DATA_BLOCK "DB00800_St_K_AnData"   // DB800
TITLE = Static DB [CONSTANTS] — Analog Card Ranges, Types and Coefficients
{ S7_Optimized_Access := 'TRUE' }
AUTHOR : M_Gledhill
FAMILY : Constants
NAME : St_K_AnData
VERSION : 0.1
// PRACTICAL SERIES AUTOMATION LIBRARY (PAL)   —   COPYRIGHT 2020 – M. GLEDHILL (MIT LICENCE)
//                   ———— ◆ ————
// FULL ONLINE DOCUMENTATION IS AVAILABLE AT: https://practicalseries.com/2001-pal/index.html
// stored: AutoNumber false, DBAccessibleFromOPCUA true, IsOnlyStoredInLoadMemory false, IsRetainMemResEnabled false, IsWriteProtectedInAS true, MemoryReserve 100
   VAR
      _DB_Header { ExternalAccessible := 'False'; ExternalVisible := 'False'; ExternalWritable := 'False'} : Array[0..79] of Bool;   // Static DB [CONSTANTS] — Analog Card Ranges, Types and Coefficients
      __________0000_0 { ExternalAccessible := 'False'; ExternalVisible := 'False'; ExternalWritable := 'False'} : Bool := false;
      __________0000_1 { ExternalAccessible := 'False'; ExternalVisible := 'False'; ExternalWritable := 'False'} : Bool := false;   // ▀▀▀▀ DB CURRENT REVISION
      revInfo { ExternalWritable := 'False'; S7_SetPoint := 'True'} : "UT01000_St_SysRevision";   // Revision information
      __________0010_0 { ExternalAccessible := 'False'; ExternalVisible := 'False'; ExternalWritable := 'False'} : Bool := false;
      __________0010_1 { ExternalAccessible := 'False'; ExternalVisible := 'False'; ExternalWritable := 'False'} : Bool := false;   // ▀▀▀▀ ANALOG SIGNAL — USER DEFINED
      AIO_0000 : "UT00800_St_K_AnData";   // User defined signal type
      __________0020_0 { ExternalAccessible := 'False'; ExternalVisible := 'False'; ExternalWritable := 'False'} : Bool := false;
      __________0020_1 { ExternalAccessible := 'False'; ExternalVisible := 'False'; ExternalWritable := 'False'} : Bool := false;   // ▀▀▀▀ ANALOG SIGNAL — VOLTAGE
      AIO_1000 : "UT00800_St_K_AnData";   // Voltage (-25 mV to +25 mV)
      AIO_1001 : "UT00800_St_K_AnData";   // Voltage (-50 mV to +50 mV)
      AIO_1002 : "UT00800_St_K_AnData";   // Voltage (-80 mV to +80 mV)
      AIO_1003 : "UT00800_St_K_AnData";   // Voltage (-250 mV to +250 mV)
      AIO_1004 : "UT00800_St_K_AnData";   // Voltage (-500 mV to +500 mV)
      AIO_1005 : "UT00800_St_K_AnData";   // Voltage (-1 V to +1 V)
      AIO_1007 : "UT00800_St_K_AnData";   // Voltage (-2.5 V to +2.5 V)
      AIO_1008 : "UT00800_St_K_AnData";   // Voltage (-5 V to +5 V)
      AIO_1009 : "UT00800_St_K_AnData";   // Voltage (-10 V to +10 V)
      AIO_100A : "UT00800_St_K_AnData";   // Voltage (1 V to 5 V)
      __________0030_0 { ExternalAccessible := 'False'; ExternalVisible := 'False'; ExternalWritable := 'False'} : Bool := false;
      __________0030_1 { ExternalAccessible := 'False'; ExternalVisible := 'False'; ExternalWritable := 'False'} : Bool := false;   // ▀▀▀▀ ANALOG SIGNAL — CURRENT (4 WIRE)
      AIO_2002 : "UT00800_St_K_AnData";   // Current - 4 wire (0 mA to 20 mA)
      AIO_2003 : "UT00800_St_K_AnData";   // Current - 4 wire (4 mA to 20 mA)
      AIO_2004 : "UT00800_St_K_AnData";   // Current - 4 wire (-20 mA to +20 mA)
      __________0040_0 { ExternalAccessible := 'False'; ExternalVisible := 'False'; ExternalWritable := 'False'} : Bool := false;
      __________0040_1 { ExternalAccessible := 'False'; ExternalVisible := 'False'; ExternalWritable := 'False'} : Bool := false;   // ▀▀▀▀ ANALOG SIGNAL — CURRENT (2 WIRE)
      AIO_3003 : "UT00800_St_K_AnData";   // Current - 2 wire (4 mA to 20 mA)
      __________0050_0 { ExternalAccessible := 'False'; ExternalVisible := 'False'; ExternalWritable := 'False'} : Bool := false;
      __________0050_1 { ExternalAccessible := 'False'; ExternalVisible := 'False'; ExternalWritable := 'False'} : Bool := false;   // ▀▀▀▀ ANALOG SIGNAL — RESISTANCE (4 WIRE)
      AIO_4001 : "UT00800_St_K_AnData";   // Resistance - 4 wire (150 Ω)
      AIO_4002 : "UT00800_St_K_AnData";   // Resistance - 4 wire (300 Ohm)
      AIO_4003 : "UT00800_St_K_AnData";   // Resistance - 4 wire (600 Ohm)
      AIO_4005 : "UT00800_St_K_AnData";   // Resistance - 4 wire (6000 Ohm)
      __________0060_0 { ExternalAccessible := 'False'; ExternalVisible := 'False'; ExternalWritable := 'False'} : Bool := false;
      __________0060_1 { ExternalAccessible := 'False'; ExternalVisible := 'False'; ExternalWritable := 'False'} : Bool := false;   // ▀▀▀▀ ANALOG SIGNAL — RESISTANCE (3 WIRE)
      AIO_5001 : "UT00800_St_K_AnData";   // Resistance - 3 wire (150 Ohm)
      AIO_5002 : "UT00800_St_K_AnData";   // Resistance - 3 wire (300 Ohm)
      AIO_5003 : "UT00800_St_K_AnData";   // Resistance - 3 wire (600 Ohm)
      AIO_5005 : "UT00800_St_K_AnData";   // Resistance - 3 wire (6000 Ohm)
      __________0070_0 { ExternalAccessible := 'False'; ExternalVisible := 'False'; ExternalWritable := 'False'} : Bool := false;
      __________0070_1 { ExternalAccessible := 'False'; ExternalVisible := 'False'; ExternalWritable := 'False'} : Bool := false;   // ▀▀▀▀ ANALOG SIGNAL — RESISTANCE (2 WIRE)
      AIO_6001 : "UT00800_St_K_AnData";   // Resistance - 2 wire (150 Ohm)
      AIO_6002 : "UT00800_St_K_AnData";   // Resistance - 2 wire (300 Ohm)
      AIO_6003 : "UT00800_St_K_AnData";   // Resistance - 2 wire (600 Ohm)
      AIO_6005 : "UT00800_St_K_AnData";   // Resistance - 2 wire (6000 Ohm)
      AIO_600F : "UT00800_St_K_AnData";   // Resistance - 2 wire (PTC)
      __________0080_0 { ExternalAccessible := 'False'; ExternalVisible := 'False'; ExternalWritable := 'False'} : Bool := false;
      __________0080_1 { ExternalAccessible := 'False'; ExternalVisible := 'False'; ExternalWritable := 'False'} : Bool := false;   // ▀▀▀▀ ANALOG SIGNAL — THERMAL RESISTANCE (4 WIRE) Cu x0
      AIO_7B0E : "UT00800_St_K_AnData";   // Thermal Resistance - 4 wire (Cu10 climate - 426)
      AIO_7C0E : "UT00800_St_K_AnData";   // Thermal Resistance - 4 wire (Cu10 climate - 427)
      AIO_7D0E : "UT00800_St_K_AnData";   // Thermal Resistance - 4 wire (Cu10 climate - 428)
      AIO_7B0F : "UT00800_St_K_AnData";   // Thermal Resistance - 4 wire (Cu10 standard - 426)
      AIO_7C0F : "UT00800_St_K_AnData";   // Thermal Resistance - 4 wire (Cu10 standard - 427)
      AIO_7D0F : "UT00800_St_K_AnData";   // Thermal Resistance - 4 wire (Cu10 standard - 428)
      AIO_7B19 : "UT00800_St_K_AnData";   // Thermal Resistance - 4 wire (Cu50 climate - 426)
      AIO_7C19 : "UT00800_St_K_AnData";   // Thermal Resistance - 4 wire (Cu50 climate - 427)
      AIO_7D19 : "UT00800_St_K_AnData";   // Thermal Resistance - 4 wire (Cu50 climate - 428)
      AIO_7B18 : "UT00800_St_K_AnData";   // Thermal Resistance - 4 wire (Cu50 standard - 426)
      AIO_7C18 : "UT00800_St_K_AnData";   // Thermal Resistance - 4 wire (Cu50 standard - 427)
      AIO_7D18 : "UT00800_St_K_AnData";   // Thermal Resistance - 4 wire (Cu50 standard - 428)
      AIO_7B1B : "UT00800_St_K_AnData";   // Thermal Resistance - 4 wire (Cu100 climate - 426)
      AIO_7C1B : "UT00800_St_K_AnData";   // Thermal Resistance - 4 wire (Cu100 climate - 427)
      AIO_7D1B : "UT00800_St_K_AnData";   // Thermal Resistance - 4 wire (Cu100 climate - 428)
      AIO_7B1A : "UT00800_St_K_AnData";   // Thermal Resistance - 4 wire (Cu100 standard - 426)
      AIO_7C1A : "UT00800_St_K_AnData";   // Thermal Resistance - 4 wire (Cu100 standard - 427)
      AIO_7D1A : "UT00800_St_K_AnData";   // Thermal Resistance - 4 wire (Cu100 standard - 428)
      __________0090_0 { ExternalAccessible := 'False'; ExternalVisible := 'False'; ExternalWritable := 'False'} : Bool := false;
      __________0090_1 { ExternalAccessible := 'False'; ExternalVisible := 'False'; ExternalWritable := 'False'} : Bool := false;   // ▀▀▀▀ ANALOG SIGNAL — THERMAL RESISTANCE (4 WIRE) LG-Ni x0
      AIO_7A1D : "UT00800_St_K_AnData";   // Thermal Resistance - 4 wire (LG-Ni1000 climate - 500)
      AIO_7A1C : "UT00800_St_K_AnData";   // Thermal Resistance - 4 wire (LG-Ni1000 standard - 500)
      __________0100_0 { ExternalAccessible := 'False'; ExternalVisible := 'False'; ExternalWritable := 'False'} : Bool := false;
      __________0100_1 { ExternalAccessible := 'False'; ExternalVisible := 'False'; ExternalWritable := 'False'} : Bool := false;   // ▀▀▀▀ ANALOG SIGNAL — THERMAL RESISTANCE (4 WIRE) Ni x0
      AIO_771F : "UT00800_St_K_AnData";   // Thermal Resistance - 4 wire (Ni10 climate - 617)
      AIO_781F : "UT00800_St_K_AnData";   // Thermal Resistance - 4 wire (Ni10 climate - 618)
      AIO_791F : "UT00800_St_K_AnData";   // Thermal Resistance - 4 wire (Ni10 climate - 672)
      AIO_771E : "UT00800_St_K_AnData";   // Thermal Resistance - 4 wire (Ni10 standard - 617)
      AIO_781E : "UT00800_St_K_AnData";   // Thermal Resistance - 4 wire (Ni10 standard - 618)
      AIO_791E : "UT00800_St_K_AnData";   // Thermal Resistance - 4 wire (Ni10 standard - 672)
      AIO_770D : "UT00800_St_K_AnData";   // Thermal Resistance - 4 wire (Ni120 climate - 617)
      AIO_780D : "UT00800_St_K_AnData";   // Thermal Resistance - 4 wire (Ni120 climate - 618)
      AIO_790D : "UT00800_St_K_AnData";   // Thermal Resistance - 4 wire (Ni120 climate - 672)
      AIO_770C : "UT00800_St_K_AnData";   // Thermal Resistance - 4 wire (Ni120 standard - 617)
      AIO_780C : "UT00800_St_K_AnData";   // Thermal Resistance - 4 wire (Ni120 standard - 618)
      AIO_790C : "UT00800_St_K_AnData";   // Thermal Resistance - 4 wire (Ni120 standard - 672)
      AIO_7701 : "UT00800_St_K_AnData";   // Thermal Resistance - 4 wire (Ni100 climate - 617)
      AIO_7801 : "UT00800_St_K_AnData";   // Thermal Resistance - 4 wire (Ni100 climate - 618)
      AIO_7901 : "UT00800_St_K_AnData";   // Thermal Resistance - 4 wire (Ni100 climate - 672)
      AIO_7703 : "UT00800_St_K_AnData";   // Thermal Resistance - 4 wire (Ni100 standard - 617)
      AIO_7803 : "UT00800_St_K_AnData";   // Thermal Resistance - 4 wire (Ni100 standard - 618)
      AIO_7903 : "UT00800_St_K_AnData";   // Thermal Resistance - 4 wire (Ni100 standard - 672)
      AIO_7711 : "UT00800_St_K_AnData";   // Thermal Resistance - 4 wire (Ni200 climate - 617)
      AIO_7811 : "UT00800_St_K_AnData";   // Thermal Resistance - 4 wire (Ni200 climate - 618)
      AIO_7911 : "UT00800_St_K_AnData";   // Thermal Resistance - 4 wire (Ni200 climate - 672)
      AIO_7710 : "UT00800_St_K_AnData";   // Thermal Resistance - 4 wire (Ni200 standard - 617)
      AIO_7810 : "UT00800_St_K_AnData";   // Thermal Resistance - 4 wire (Ni200 standard - 618)
      AIO_7910 : "UT00800_St_K_AnData";   // Thermal Resistance - 4 wire (Ni200 standard - 672)
      AIO_7713 : "UT00800_St_K_AnData";   // Thermal Resistance - 4 wire (Ni500 climate - 617)
      AIO_7813 : "UT00800_St_K_AnData";   // Thermal Resistance - 4 wire (Ni500 climate - 618)
      AIO_7913 : "UT00800_St_K_AnData";   // Thermal Resistance - 4 wire (Ni500 climate - 672)
      AIO_7712 : "UT00800_St_K_AnData";   // Thermal Resistance - 4 wire (Ni500 standard - 617)
      AIO_7812 : "UT00800_St_K_AnData";   // Thermal Resistance - 4 wire (Ni500 standard - 618)
      AIO_7912 : "UT00800_St_K_AnData";   // Thermal Resistance - 4 wire (Ni500 standard - 672)
      AIO_770A : "UT00800_St_K_AnData";   // Thermal Resistance - 4 wire (Ni1000 climate - 617)
      AIO_780A : "UT00800_St_K_AnData";   // Thermal Resistance - 4 wire (Ni1000 climate - 618)
      AIO_790A : "UT00800_St_K_AnData";   // Thermal Resistance - 4 wire (Ni1000 climate - 672)
      AIO_7706 : "UT00800_St_K_AnData";   // Thermal Resistance - 4 wire (Ni1000 standard - 617)
      AIO_7806 : "UT00800_St_K_AnData";   // Thermal Resistance - 4 wire (Ni1000 standard - 618)
      AIO_7906 : "UT00800_St_K_AnData";   // Thermal Resistance - 4 wire (Ni1000 standard - 672)
      __________0110_0 { ExternalAccessible := 'False'; ExternalVisible := 'False'; ExternalWritable := 'False'} : Bool := false;
      __________0110_1 { ExternalAccessible := 'False'; ExternalVisible := 'False'; ExternalWritable := 'False'} : Bool := false;   // ▀▀▀▀ ANALOG SIGNAL — THERMAL RESISTANCE (4 WIRE) Pt x0
      AIO_7015 : "UT00800_St_K_AnData";   // Thermal Resistance - 4 wire (Pt10 climate - 3851)
      AIO_7215 : "UT00800_St_K_AnData";   // Thermal Resistance - 4 wire (Pt10 climate - 3902)
      AIO_7515 : "UT00800_St_K_AnData";   // Thermal Resistance - 4 wire (Pt10 climate - 391)
      AIO_7115 : "UT00800_St_K_AnData";   // Thermal Resistance - 4 wire (Pt10 climate - 3916)
      AIO_7315 : "UT00800_St_K_AnData";   // Thermal Resistance - 4 wire (Pt10 climate - 392)
      AIO_7014 : "UT00800_St_K_AnData";   // Thermal Resistance - 4 wire (Pt10 standard - 3851)
      AIO_7214 : "UT00800_St_K_AnData";   // Thermal Resistance - 4 wire (Pt10 standard - 3902)
      AIO_7514 : "UT00800_St_K_AnData";   // Thermal Resistance - 4 wire (Pt10 standard - 391)
      AIO_7114 : "UT00800_St_K_AnData";   // Thermal Resistance - 4 wire (Pt10 standard - 3916)
      AIO_7314 : "UT00800_St_K_AnData";   // Thermal Resistance - 4 wire (Pt10 standard - 392)
      AIO_7017 : "UT00800_St_K_AnData";   // Thermal Resistance - 4 wire (Pt50 climate - 3851)
      AIO_7217 : "UT00800_St_K_AnData";   // Thermal Resistance - 4 wire (Pt50 climate - 3902)
      AIO_7517 : "UT00800_St_K_AnData";   // Thermal Resistance - 4 wire (Pt50 climate - 391)
      AIO_7117 : "UT00800_St_K_AnData";   // Thermal Resistance - 4 wire (Pt50 climate - 3916)
      AIO_7317 : "UT00800_St_K_AnData";   // Thermal Resistance - 4 wire (Pt50 climate - 392)
      AIO_7016 : "UT00800_St_K_AnData";   // Thermal Resistance - 4 wire (Pt50 standard - 3851)
      AIO_7216 : "UT00800_St_K_AnData";   // Thermal Resistance - 4 wire (Pt50 standard - 3902)
      AIO_7516 : "UT00800_St_K_AnData";   // Thermal Resistance - 4 wire (Pt50 standard - 391)
      AIO_7116 : "UT00800_St_K_AnData";   // Thermal Resistance - 4 wire (Pt50 standard - 3916)
      AIO_7316 : "UT00800_St_K_AnData";   // Thermal Resistance - 4 wire (Pt50 standard - 392)
      AIO_7000 : "UT00800_St_K_AnData";   // Thermal Resistance - 4 wire (Pt100 climate - 3851)
      AIO_7200 : "UT00800_St_K_AnData";   // Thermal Resistance - 4 wire (Pt100 climate - 3902)
      AIO_7500 : "UT00800_St_K_AnData";   // Thermal Resistance - 4 wire (Pt100 climate - 391)
      AIO_7100 : "UT00800_St_K_AnData";   // Thermal Resistance - 4 wire (Pt100 climate - 3916)
      AIO_7300 : "UT00800_St_K_AnData";   // Thermal Resistance - 4 wire (Pt100 climate - 392)
      AIO_7002 : "UT00800_St_K_AnData";   // Thermal Resistance - 4 wire (Pt100 standard - 3851)
      AIO_7202 : "UT00800_St_K_AnData";   // Thermal Resistance - 4 wire (Pt100 standard - 3902)
      AIO_7502 : "UT00800_St_K_AnData";   // Thermal Resistance - 4 wire (Pt100 standard - 391)
      AIO_7102 : "UT00800_St_K_AnData";   // Thermal Resistance - 4 wire (Pt100 standard - 3916)
      AIO_7302 : "UT00800_St_K_AnData";   // Thermal Resistance - 4 wire (Pt100 standard - 392)
      AIO_7007 : "UT00800_St_K_AnData";   // Thermal Resistance - 4 wire (Pt200 climate - 3851)
      AIO_7207 : "UT00800_St_K_AnData";   // Thermal Resistance - 4 wire (Pt200 climate - 3902)
      AIO_7507 : "UT00800_St_K_AnData";   // Thermal Resistance - 4 wire (Pt200 climate - 391)
      AIO_7107 : "UT00800_St_K_AnData";   // Thermal Resistance - 4 wire (Pt200 climate - 3916)
      AIO_7307 : "UT00800_St_K_AnData";   // Thermal Resistance - 4 wire (Pt200 climate - 392)
      AIO_700B : "UT00800_St_K_AnData";   // Thermal Resistance - 4 wire (Pt200 standard - 3851)
      AIO_720B : "UT00800_St_K_AnData";   // Thermal Resistance - 4 wire (Pt200 standard - 3902)
      AIO_750B : "UT00800_St_K_AnData";   // Thermal Resistance - 4 wire (Pt200 standard - 391)
      AIO_710B : "UT00800_St_K_AnData";   // Thermal Resistance - 4 wire (Pt200 standard - 3916)
      AIO_730B : "UT00800_St_K_AnData";   // Thermal Resistance - 4 wire (Pt200 standard - 392)
      AIO_7008 : "UT00800_St_K_AnData";   // Thermal Resistance - 4 wire (Pt500 climate - 3851)
      AIO_7208 : "UT00800_St_K_AnData";   // Thermal Resistance - 4 wire (Pt500 climate - 3902)
      AIO_7508 : "UT00800_St_K_AnData";   // Thermal Resistance - 4 wire (Pt500 climate - 3902)
      AIO_7108 : "UT00800_St_K_AnData";   // Thermal Resistance - 4 wire (Pt500 climate - 3916)
      AIO_7308 : "UT00800_St_K_AnData";   // Thermal Resistance - 4 wire (Pt500 climate - 392)
      AIO_7004 : "UT00800_St_K_AnData";   // Thermal Resistance - 4 wire (Pt500 standard - 3851)
      AIO_7204 : "UT00800_St_K_AnData";   // Thermal Resistance - 4 wire (Pt500 standard - 3902)
      AIO_7504 : "UT00800_St_K_AnData";   // Thermal Resistance - 4 wire (Pt500 standard - 391)
      AIO_7104 : "UT00800_St_K_AnData";   // Thermal Resistance - 4 wire (Pt500 standard - 3916)
      AIO_7304 : "UT00800_St_K_AnData";   // Thermal Resistance - 4 wire (Pt500 standard - 392)
      AIO_7009 : "UT00800_St_K_AnData";   // Thermal Resistance - 4 wire (Pt1000 climate - 3851)
      AIO_7209 : "UT00800_St_K_AnData";   // Thermal Resistance - 4 wire (Pt1000 climate - 3902)
      AIO_7509 : "UT00800_St_K_AnData";   // Thermal Resistance - 4 wire (Pt1000 climate - 391)
      AIO_7109 : "UT00800_St_K_AnData";   // Thermal Resistance - 4 wire (Pt1000 climate - 3916)
      AIO_7309 : "UT00800_St_K_AnData";   // Thermal Resistance - 4 wire (Pt1000 climate - 392)
      AIO_7005 : "UT00800_St_K_AnData";   // Thermal Resistance - 4 wire (Pt1000 standard - 3851)
      AIO_7205 : "UT00800_St_K_AnData";   // Thermal Resistance - 4 wire (Pt1000 standard - 3902)
      AIO_7505 : "UT00800_St_K_AnData";   // Thermal Resistance - 4 wire (Pt1000 standard - 391)
      AIO_7105 : "UT00800_St_K_AnData";   // Thermal Resistance - 4 wire (Pt1000 standard - 3916)
      AIO_7305 : "UT00800_St_K_AnData";   // Thermal Resistance - 4 wire (Pt1000 standard - 392)
      "199" : "UT00800_St_K_AnData";   // Voltage — -10 V to 10 V
      __________0120_0 { ExternalAccessible := 'False'; ExternalVisible := 'False'; ExternalWritable := 'False'} : Bool := false;
      __________0120_1 { ExternalAccessible := 'False'; ExternalVisible := 'False'; ExternalWritable := 'False'} : Bool := false;   // ▀▀▀▀ ANALOG SIGNAL — THERMAL RESISTANCE (3 WIRE) Cu x0
      AIO_8B0E : "UT00800_St_K_AnData";   // Thermal Resistance - 3-wire (Cu10 climate - 426)
      AIO_8C0E : "UT00800_St_K_AnData";   // Thermal Resistance - 3-wire (Cu10 climate - 427)
      AIO_8D0E : "UT00800_St_K_AnData";   // Thermal Resistance - 3-wire (Cu10 climate - 428)
      AIO_8B0F : "UT00800_St_K_AnData";   // Thermal Resistance - 3-wire (Cu10 standard - 426)
      AIO_8C0F : "UT00800_St_K_AnData";   // Thermal Resistance - 3-wire (Cu10 standard - 427)
      AIO_8D0F : "UT00800_St_K_AnData";   // Thermal Resistance - 3-wire (Cu10 standard - 428)
      AIO_8B19 : "UT00800_St_K_AnData";   // Thermal Resistance - 3-wire (Cu50 climate - 426)
      AIO_8C19 : "UT00800_St_K_AnData";   // Thermal Resistance - 3-wire (Cu50 climate - 427)
      AIO_8D19 : "UT00800_St_K_AnData";   // Thermal Resistance - 3-wire (Cu50 climate - 428)
      AIO_8B18 : "UT00800_St_K_AnData";   // Thermal Resistance - 3-wire (Cu50 standard - 426)
      AIO_8C18 : "UT00800_St_K_AnData";   // Thermal Resistance - 3-wire (Cu50 standard - 427)
      AIO_8D18 : "UT00800_St_K_AnData";   // Thermal Resistance - 3-wire (Cu50 standard - 428)
      AIO_8B1B : "UT00800_St_K_AnData";   // Thermal Resistance - 3-wire (Cu100 climate - 426)
      AIO_8C1B : "UT00800_St_K_AnData";   // Thermal Resistance - 3-wire (Cu100 climate - 427)
      AIO_8D1B : "UT00800_St_K_AnData";   // Thermal Resistance - 3-wire (Cu100 climate - 428)
      AIO_8B1A : "UT00800_St_K_AnData";   // Thermal Resistance - 3-wire (Cu100 standard - 426)
      AIO_8C1A : "UT00800_St_K_AnData";   // Thermal Resistance - 3-wire (Cu100 standard - 427)
      AIO_8D1A : "UT00800_St_K_AnData";   // Thermal Resistance - 3-wire (Cu100 standard - 428)
      __________0130_0 { ExternalAccessible := 'False'; ExternalVisible := 'False'; ExternalWritable := 'False'} : Bool := false;
      __________0130_1 { ExternalAccessible := 'False'; ExternalVisible := 'False'; ExternalWritable := 'False'} : Bool := false;   // ▀▀▀▀ ANALOG SIGNAL — THERMAL RESISTANCE (3 WIRE) LG-Ni x0
      AIO_8A1D : "UT00800_St_K_AnData";   // Thermal Resistance - 3-wire (LG-Ni1000 climate - 500)
      AIO_8A1C : "UT00800_St_K_AnData";   // Thermal Resistance - 3-wire (LG-Ni1000 standard - 500)
      __________0140_0 { ExternalAccessible := 'False'; ExternalVisible := 'False'; ExternalWritable := 'False'} : Bool := false;
      __________0140_1 { ExternalAccessible := 'False'; ExternalVisible := 'False'; ExternalWritable := 'False'} : Bool := false;   // ▀▀▀▀ ANALOG SIGNAL — THERMAL RESISTANCE (3 WIRE) Ni x0
      AIO_871F : "UT00800_St_K_AnData";   // Thermal Resistance - 3-wire (Ni10 climate - 617)
      AIO_881F : "UT00800_St_K_AnData";   // Thermal Resistance - 3-wire (Ni10 climate - 618)
      AIO_891F : "UT00800_St_K_AnData";   // Thermal Resistance - 3-wire (Ni10 climate - 672)
      AIO_871E : "UT00800_St_K_AnData";   // Thermal Resistance - 3-wire (Ni10 standard - 617)
      AIO_881E : "UT00800_St_K_AnData";   // Thermal Resistance - 3-wire (Ni10 standard - 618)
      AIO_891E : "UT00800_St_K_AnData";   // Thermal Resistance - 3-wire (Ni10 standard - 672)
      AIO_870D : "UT00800_St_K_AnData";   // Thermal Resistance - 3-wire (Ni120 climate - 617)
      AIO_880D : "UT00800_St_K_AnData";   // Thermal Resistance - 3-wire (Ni120 climate - 618)
      AIO_890D : "UT00800_St_K_AnData";   // Thermal Resistance - 3-wire (Ni120 climate - 672)
      AIO_870C : "UT00800_St_K_AnData";   // Thermal Resistance - 3-wire (Ni120 standard - 617)
      AIO_880C : "UT00800_St_K_AnData";   // Thermal Resistance - 3-wire (Ni120 standard - 618)
      AIO_890C : "UT00800_St_K_AnData";   // Thermal Resistance - 3-wire (Ni120 standard - 672)
      AIO_8701 : "UT00800_St_K_AnData";   // Thermal Resistance - 3-wire (Ni100 climate - 617)
      AIO_8801 : "UT00800_St_K_AnData";   // Thermal Resistance - 3-wire (Ni100 climate - 618)
      AIO_8901 : "UT00800_St_K_AnData";   // Thermal Resistance - 3-wire (Ni100 climate - 672)
      AIO_8703 : "UT00800_St_K_AnData";   // Thermal Resistance - 3-wire (Ni100 standard - 617)
      AIO_8803 : "UT00800_St_K_AnData";   // Thermal Resistance - 3-wire (Ni100 standard - 618)
      AIO_8903 : "UT00800_St_K_AnData";   // Thermal Resistance - 3-wire (Ni100 standard - 672)
      AIO_8711 : "UT00800_St_K_AnData";   // Thermal Resistance - 3-wire (Ni200 climate - 617)
      AIO_8811 : "UT00800_St_K_AnData";   // Thermal Resistance - 3-wire (Ni200 climate - 618)
      AIO_8911 : "UT00800_St_K_AnData";   // Thermal Resistance - 3-wire (Ni200 climate - 672)
      AIO_8710 : "UT00800_St_K_AnData";   // Thermal Resistance - 3-wire (Ni200 standard - 617)
      AIO_8810 : "UT00800_St_K_AnData";   // Thermal Resistance - 3-wire (Ni200 standard - 618)
      AIO_8910 : "UT00800_St_K_AnData";   // Thermal Resistance - 3-wire (Ni200 standard - 672)
      AIO_8713 : "UT00800_St_K_AnData";   // Thermal Resistance - 3-wire (Ni500 climate - 617)
      AIO_8813 : "UT00800_St_K_AnData";   // Thermal Resistance - 3-wire (Ni500 climate - 618)
      AIO_8913 : "UT00800_St_K_AnData";   // Thermal Resistance - 3-wire (Ni500 climate - 672)
      AIO_8712 : "UT00800_St_K_AnData";   // Thermal Resistance - 3-wire (Ni500 standard - 617)
      AIO_8812 : "UT00800_St_K_AnData";   // Thermal Resistance - 3-wire (Ni500 standard - 618)
      AIO_8912 : "UT00800_St_K_AnData";   // Thermal Resistance - 3-wire (Ni500 standard - 672)
      AIO_870A : "UT00800_St_K_AnData";   // Thermal Resistance - 3-wire (Ni1000 climate - 617)
      AIO_880A : "UT00800_St_K_AnData";   // Thermal Resistance - 3-wire (Ni1000 climate - 618)
      AIO_890A : "UT00800_St_K_AnData";   // Thermal Resistance - 3-wire (Ni1000 climate - 672)
      AIO_8706 : "UT00800_St_K_AnData";   // Thermal Resistance - 3-wire (Ni1000 standard - 617)
      AIO_8806 : "UT00800_St_K_AnData";   // Thermal Resistance - 3-wire (Ni1000 standard - 618)
      AIO_8906 : "UT00800_St_K_AnData";   // Thermal Resistance - 3-wire (Ni1000 standard - 672)
      __________0150_0 { ExternalAccessible := 'False'; ExternalVisible := 'False'; ExternalWritable := 'False'} : Bool := false;
      __________0150_1 { ExternalAccessible := 'False'; ExternalVisible := 'False'; ExternalWritable := 'False'} : Bool := false;   // ▀▀▀▀ ANALOG SIGNAL — THERMAL RESISTANCE (3 WIRE) Pt x0
      AIO_8015 : "UT00800_St_K_AnData";   // Thermal Resistance - 3-wire (Pt10 climate - 3851)
      AIO_8215 : "UT00800_St_K_AnData";   // Thermal Resistance - 3-wire (Pt10 climate - 3902)
      AIO_8515 : "UT00800_St_K_AnData";   // Thermal Resistance - 3-wire (Pt10 climate - 391)
      AIO_8115 : "UT00800_St_K_AnData";   // Thermal Resistance - 3-wire (Pt10 climate - 3916)
      AIO_8315 : "UT00800_St_K_AnData";   // Thermal Resistance - 3-wire (Pt10 climate - 392)
      AIO_8014 : "UT00800_St_K_AnData";   // Thermal Resistance - 3-wire (Pt10 standard - 3851)
      AIO_8214 : "UT00800_St_K_AnData";   // Thermal Resistance - 3-wire (Pt10 standard - 3902)
      AIO_8514 : "UT00800_St_K_AnData";   // Thermal Resistance - 3-wire (Pt10 standard - 391)
      AIO_8114 : "UT00800_St_K_AnData";   // Thermal Resistance - 3-wire (Pt10 standard - 3916)
      AIO_8314 : "UT00800_St_K_AnData";   // Thermal Resistance - 3-wire (Pt10 standard - 392)
      AIO_8017 : "UT00800_St_K_AnData";   // Thermal Resistance - 3-wire (Pt50 climate - 3851)
      AIO_8217 : "UT00800_St_K_AnData";   // Thermal Resistance - 3-wire (Pt50 climate - 3902)
      AIO_8517 : "UT00800_St_K_AnData";   // Thermal Resistance - 3-wire (Pt50 climate - 391)
      AIO_8117 : "UT00800_St_K_AnData";   // Thermal Resistance - 3-wire (Pt50 climate - 3916)
      AIO_8317 : "UT00800_St_K_AnData";   // Thermal Resistance - 3-wire (Pt50 climate - 392)
      AIO_8016 : "UT00800_St_K_AnData";   // Thermal Resistance - 3-wire (Pt50 standard - 3851)
      AIO_8216 : "UT00800_St_K_AnData";   // Thermal Resistance - 3-wire (Pt50 standard - 3902)
      AIO_8516 : "UT00800_St_K_AnData";   // Thermal Resistance - 3-wire (Pt50 standard - 391)
      AIO_8116 : "UT00800_St_K_AnData";   // Thermal Resistance - 3-wire (Pt50 standard - 3916)
      AIO_8316 : "UT00800_St_K_AnData";   // Thermal Resistance - 3-wire (Pt50 standard - 392)
      AIO_8000 : "UT00800_St_K_AnData";   // Thermal Resistance - 3-wire (Pt100 climate - 3851)
      AIO_8200 : "UT00800_St_K_AnData";   // Thermal Resistance - 3-wire (Pt100 climate - 3902)
      AIO_8500 : "UT00800_St_K_AnData";   // Thermal Resistance - 3-wire (Pt100 climate - 391)
      AIO_8100 : "UT00800_St_K_AnData";   // Thermal Resistance - 3-wire (Pt100 climate - 3916)
      AIO_8300 { S7_SetPoint := 'True'} : "UT00800_St_K_AnData";   // Thermal Resistance - 3-wire (Pt100 climate - 392)
      AIO_8002 : "UT00800_St_K_AnData";   // Thermal Resistance - 3-wire (Pt100 standard - 3851)
      AIO_8202 : "UT00800_St_K_AnData";   // Thermal Resistance - 3-wire (Pt100 standard - 3902)
      AIO_8502 : "UT00800_St_K_AnData";   // Thermal Resistance - 3-wire (Pt100 standard - 391)
      AIO_8102 : "UT00800_St_K_AnData";   // Thermal Resistance - 3-wire (Pt100 standard - 3916)
      AIO_8302 : "UT00800_St_K_AnData";   // Thermal Resistance - 3-wire (Pt100 standard - 392)
      AIO_8007 : "UT00800_St_K_AnData";   // Thermal Resistance - 3-wire (Pt200 climate - 3851)
      AIO_8207 : "UT00800_St_K_AnData";   // Thermal Resistance - 3-wire (Pt200 climate - 3902)
      AIO_8507 : "UT00800_St_K_AnData";   // Thermal Resistance - 3-wire (Pt200 climate - 391)
      AIO_8107 : "UT00800_St_K_AnData";   // Thermal Resistance - 3-wire (Pt200 climate - 3916)
      AIO_8307 : "UT00800_St_K_AnData";   // Thermal Resistance - 3-wire (Pt200 climate - 392)
      AIO_800B : "UT00800_St_K_AnData";   // Thermal Resistance - 3-wire (Pt200 standard - 3851)
      AIO_820B : "UT00800_St_K_AnData";   // Thermal Resistance - 3-wire (Pt200 standard - 3902)
      AIO_850B : "UT00800_St_K_AnData";   // Thermal Resistance - 3-wire (Pt200 standard - 391)
      AIO_810B : "UT00800_St_K_AnData";   // Thermal Resistance - 3-wire (Pt200 standard - 3916)
      AIO_830B : "UT00800_St_K_AnData";   // Thermal Resistance - 3-wire (Pt200 standard - 392)
      AIO_8008 : "UT00800_St_K_AnData";   // Thermal Resistance - 3-wire (Pt500 climate - 3851)
      AIO_8208 : "UT00800_St_K_AnData";   // Thermal Resistance - 3-wire (Pt500 climate - 3902)
      AIO_8508 : "UT00800_St_K_AnData";   // Thermal Resistance - 3-wire (Pt500 climate - 3902)
      AIO_8108 : "UT00800_St_K_AnData";   // Thermal Resistance - 3-wire (Pt500 climate - 3916)
      AIO_8308 : "UT00800_St_K_AnData";   // Thermal Resistance - 3-wire (Pt500 climate - 392)
      AIO_8004 : "UT00800_St_K_AnData";   // Thermal Resistance - 3-wire (Pt500 standard - 3851)
      AIO_8204 : "UT00800_St_K_AnData";   // Thermal Resistance - 3-wire (Pt500 standard - 3902)
      AIO_8504 : "UT00800_St_K_AnData";   // Thermal Resistance - 3-wire (Pt500 standard - 391)
      AIO_8104 : "UT00800_St_K_AnData";   // Thermal Resistance - 3-wire (Pt500 standard - 3916)
      AIO_8304 : "UT00800_St_K_AnData";   // Thermal Resistance - 3-wire (Pt500 standard - 392)
      AIO_8009 : "UT00800_St_K_AnData";   // Thermal Resistance - 3-wire (Pt1000 climate - 3851)
      AIO_8209 : "UT00800_St_K_AnData";   // Thermal Resistance - 3-wire (Pt1000 climate - 3902)
      AIO_8509 : "UT00800_St_K_AnData";   // Thermal Resistance - 3-wire (Pt1000 climate - 391)
      AIO_8109 : "UT00800_St_K_AnData";   // Thermal Resistance - 3-wire (Pt1000 climate - 3916)
      AIO_8309 : "UT00800_St_K_AnData";   // Thermal Resistance - 3-wire (Pt1000 climate - 392)
      AIO_8005 : "UT00800_St_K_AnData";   // Thermal Resistance - 3-wire (Pt1000 standard - 3851)
      AIO_8205 : "UT00800_St_K_AnData";   // Thermal Resistance - 3-wire (Pt1000 standard - 3902)
      AIO_8505 : "UT00800_St_K_AnData";   // Thermal Resistance - 3-wire (Pt1000 standard - 391)
      AIO_8105 : "UT00800_St_K_AnData";   // Thermal Resistance - 3-wire (Pt1000 standard - 3916)
      AIO_8305 : "UT00800_St_K_AnData";   // Thermal Resistance - 3-wire (Pt1000 standard - 392)
      __________0160_0 { ExternalAccessible := 'False'; ExternalVisible := 'False'; ExternalWritable := 'False'} : Bool := false;
      __________0160_1 { ExternalAccessible := 'False'; ExternalVisible := 'False'; ExternalWritable := 'False'} : Bool := false;   // ▀▀▀▀ ANALOG SIGNAL — THERMOCOUPLE
      AIO_A000 : "UT00800_St_K_AnData";   // Thermocouple (Type B)
      AIO_A00A : "UT00800_St_K_AnData";   // Thermocouple (Type C)
      AIO_A002 : "UT00800_St_K_AnData";   // Thermocouple (Type E)
      AIO_A005 : "UT00800_St_K_AnData";   // Thermocouple (Type J)
      AIO_A008 : "UT00800_St_K_AnData";   // Thermocouple (Type K)
      AIO_A001 : "UT00800_St_K_AnData";   // Thermocouple (Type N)
      AIO_A003 : "UT00800_St_K_AnData";   // Thermocouple (Type R)
      AIO_A004 : "UT00800_St_K_AnData";   // Thermocouple (Type S)
      AIO_A007 : "UT00800_St_K_AnData";   // Thermocouple (Type T)
      AIO_A00B : "UT00800_St_K_AnData";   // Thermocouple (Type TXK/XCL)
   END_VAR
BEGIN
   // _DB_Header[0] : ▄▄▄▄▄▄▄▄▄▄▄▄▄▄▄▄▄▄▄▄▄▄▄▄▄▄▄▄▄▄▄▄ ＣＯＮＳＴＡＮＴＳ ▄▄
   // _DB_Header[2] : TITLE: CONSTANTS — ANALOG CARD RANGES, TYPES & COEFFICIENTS
   // _DB_Header[4] : ▀▀▀▀▀▀▀▀▀▀▀▀▀▀▀▀▀▀▀▀▀▀▀▀▀▀▀▀▀▀▀▀▀▀▀▀▀▀▀▀▀▀▀▀
   // _DB_Header[5] : TYPE: STATIC
   // _DB_Header[6] : ▄▄▄▄▄▄▄▄▄▄▄▄▄▄▄▄▄▄▄▄▄▄▄▄▄▄▄▄▄▄▄▄▄▄▄▄▄▄▄▄▄▄▄▄
   // _DB_Header[8] : This is a static set of constant data specifying the standard RAW_MIN and RAW_MAX ranges for
   // _DB_Header[9] : the common types of analog input: voltage, current, resistance, thermocouple and RTD
   // _DB_Header[11] : It stores the parameters that can be used to specify card ranges at run time:
   // _DB_Header[12] : PARAM_TYPE Identifies the channel type: voltage, current, resistance &c.
   // _DB_Header[13] : PARAM_RANGE Identifies the channel range: 1-5V, 4-20mA &c.
   // _DB_Header[14] : PARAM_COEF Specifies the temperature coefficient for thermal resistance channel types
   // _DB_Header[16] : The thermal coefficient is stored in full as a real number in the variable VALUE_COEF
   // _DB_Header[18] : Each valve is given the user data type:
   // _DB_Header[19] : UT00800_St_K_AnData
   // _DB_Header[20] : This holds the full set of static configuration data for each analog input type
   // _DB_Header[22] : ━━━ ⬙⬙⬙⬙⬙⬙ ━━━
   // _DB_Header[24] : ▄▄▄▄▄▄▄▄▄▄▄▄▄▄▄▄▄▄▄▄▄▄▄▄▄▄▄▄▄▄▄▄▄▄▄▄▄▄▄▄▄▄▄▄
   // _DB_Header[25] : MODIFICATION HISTORY
   // _DB_Header[27] : This is a summary of the recent software modifications made to this block (most recent at top)
   // _DB_Header[29] : ―――――――――――――――――――――――――――――――――――――――――――
   // _DB_Header[30] : DATE REVISION MASTER BRANCH DEV
   // _DB_Header[31] : (nnn.amm) COMMIT TAG (Base ---> Merge) BRANCH Author
   // _DB_Header[32] : ———————————————————————————————————————————
   // _DB_Header[33] : 2024.04.09 000.101 D0017A-000.101 D0017 N/A D0017A M. Gledhill
   // _DB_Header[34] : DB00800 Block created
   // _DB_Header[35] : ———————————————————————————————————————————
   // _DB_Header[36] : Where: nnn = Major revision
   // _DB_Header[37] : a = Type (1-7 Development, 8 Proving, 9 Qualification, 0 Release)
   // _DB_Header[38] : mm = Minor revision (must be 00 if a = 0)
   // _DB_Header[39] : Block properties version number should be set to nn.a (only one decimal place)
   // _DB_Header[41] : ██████████████ █ █ █ █ END █ █ █ █ ██████████████
   revInfo.REV_BLOCK := 'DB00800';
   revInfo.REV_NUMBER := '000.101';
   revInfo.REV_DATE := '2024-04-09';
   revInfo.REV_AUTHOR := 'M. Gledhill';
   AIO_0000.AIO_CODE := 16#0000;
   AIO_0000.___________0020_0 := false;
   AIO_0000.___________0010_2 := false;
   AIO_0000.RAW_MIN := 0;
   AIO_0000.RAW_MAX := 0;
   AIO_0000.RAW_NAME := 'User defined signal type';
   AIO_0000.___________0030_1 := false;
   AIO_0000.___________0030_2 := false;
   AIO_0000.PARAM_TYPE := 16#00;
   AIO_0000.PARAM_RANGE := 16#00;
   AIO_0000.PARAM_COEF := 16#00;
   AIO_1000.AIO_CODE := 16#1000;
   AIO_1000.___________0020_0 := false;
   AIO_1000.___________0010_2 := false;
   AIO_1000.RAW_MIN := -27648;
   AIO_1000.RAW_MAX := 27648;
   AIO_1000.RAW_NAME := 'Voltage (-25 mV to +25 mV)';
   AIO_1000.___________0030_1 := false;
   AIO_1000.___________0030_2 := false;
   AIO_1000.PARAM_TYPE := 16#01;
   AIO_1000.PARAM_RANGE := 16#00;
   AIO_1000.PARAM_COEF := 16#00;
   AIO_1001.AIO_CODE := 16#1001;
   AIO_1001.___________0020_0 := false;
   AIO_1001.___________0010_2 := false;
   AIO_1001.RAW_MIN := -27648;
   AIO_1001.RAW_MAX := 27648;
   AIO_1001.RAW_NAME := 'Voltage (-50 mV to +50 mV)';
   AIO_1001.___________0030_1 := false;
   AIO_1001.___________0030_2 := false;
   AIO_1001.PARAM_TYPE := 16#01;
   AIO_1001.PARAM_RANGE := 16#01;
   AIO_1001.PARAM_COEF := 16#00;
   AIO_1002.AIO_CODE := 16#1002;
   AIO_1002.___________0020_0 := false;
   AIO_1002.___________0010_2 := false;
   AIO_1002.RAW_MIN := -27648;
   AIO_1002.RAW_MAX := 27648;
   AIO_1002.RAW_NAME := 'Voltage (-80 mV to +80 mV)';
   AIO_1002.___________0030_1 := false;
   AIO_1002.___________0030_2 := false;
   AIO_1002.PARAM_TYPE := 16#01;
   AIO_1002.PARAM_RANGE := 16#02;
   AIO_1002.PARAM_COEF := 16#00;
   AIO_1003.AIO_CODE := 16#1003;
   AIO_1003.___________0020_0 := false;
   AIO_1003.___________0010_2 := false;
   AIO_1003.RAW_MIN := -27648;
   AIO_1003.RAW_MAX := 27648;
   AIO_1003.RAW_NAME := 'Voltage (-250 mV to +250 mV)';
   AIO_1003.___________0030_1 := false;
   AIO_1003.___________0030_2 := false;
   AIO_1003.PARAM_TYPE := 16#01;
   AIO_1003.PARAM_RANGE := 16#03;
   AIO_1003.PARAM_COEF := 16#00;
   AIO_1004.AIO_CODE := 16#1004;
   AIO_1004.___________0020_0 := false;
   AIO_1004.___________0010_2 := false;
   AIO_1004.RAW_MIN := -27648;
   AIO_1004.RAW_MAX := 27648;
   AIO_1004.RAW_NAME := 'Voltage (-500 mV to +500 mV)';
   AIO_1004.___________0030_1 := false;
   AIO_1004.___________0030_2 := false;
   AIO_1004.PARAM_TYPE := 16#01;
   AIO_1004.PARAM_RANGE := 16#04;
   AIO_1004.PARAM_COEF := 16#00;
   AIO_1005.AIO_CODE := 16#1005;
   AIO_1005.___________0020_0 := false;
   AIO_1005.___________0010_2 := false;
   AIO_1005.RAW_MIN := -27648;
   AIO_1005.RAW_MAX := 27648;
   AIO_1005.RAW_NAME := 'Voltage (-1 V to +1 V)';
   AIO_1005.___________0030_1 := false;
   AIO_1005.___________0030_2 := false;
   AIO_1005.PARAM_TYPE := 16#01;
   AIO_1005.PARAM_RANGE := 16#05;
   AIO_1005.PARAM_COEF := 16#00;
   AIO_1007.AIO_CODE := 16#1007;
   AIO_1007.___________0020_0 := false;
   AIO_1007.___________0010_2 := false;
   AIO_1007.RAW_MIN := -27648;
   AIO_1007.RAW_MAX := 27648;
   AIO_1007.RAW_NAME := 'Voltage (-2.5 V to +2.5 V)';
   AIO_1007.___________0030_1 := false;
   AIO_1007.___________0030_2 := false;
   AIO_1007.PARAM_TYPE := 16#01;
   AIO_1007.PARAM_RANGE := 16#07;
   AIO_1007.PARAM_COEF := 16#00;
   AIO_1008.AIO_CODE := 16#1008;
   AIO_1008.___________0020_0 := false;
   AIO_1008.___________0010_2 := false;
   AIO_1008.RAW_MIN := -27648;
   AIO_1008.RAW_MAX := 27648;
   AIO_1008.RAW_NAME := 'Voltage (-5 V to +5 V)';
   AIO_1008.___________0030_1 := false;
   AIO_1008.___________0030_2 := false;
   AIO_1008.PARAM_TYPE := 16#01;
   AIO_1008.PARAM_RANGE := 16#08;
   AIO_1008.PARAM_COEF := 16#00;
   AIO_1009.AIO_CODE := 16#1009;
   AIO_1009.___________0020_0 := false;
   AIO_1009.___________0010_2 := false;
   AIO_1009.RAW_MIN := -27648;
   AIO_1009.RAW_MAX := 27648;
   AIO_1009.RAW_NAME := 'Voltage (-10 V to +10 V)';
   AIO_1009.___________0030_1 := false;
   AIO_1009.___________0030_2 := false;
   AIO_1009.PARAM_TYPE := 16#01;
   AIO_1009.PARAM_RANGE := 16#09;
   AIO_1009.PARAM_COEF := 16#00;
   AIO_100A.AIO_CODE := 16#100A;
   AIO_100A.___________0020_0 := false;
   AIO_100A.___________0010_2 := false;
   AIO_100A.RAW_MIN := 0;
   AIO_100A.RAW_MAX := 27648;
   AIO_100A.RAW_NAME := 'Voltage (1 V to 5 V)';
   AIO_100A.___________0030_1 := false;
   AIO_100A.___________0030_2 := false;
   AIO_100A.PARAM_TYPE := 16#01;
   AIO_100A.PARAM_RANGE := 16#0A;
   AIO_100A.PARAM_COEF := 16#00;
   AIO_2002.AIO_CODE := 16#2002;
   AIO_2002.___________0020_0 := false;
   AIO_2002.___________0010_2 := false;
   AIO_2002.RAW_MIN := 0;
   AIO_2002.RAW_MAX := 27648;
   AIO_2002.RAW_NAME := 'Current - 4 wire (0 mA to 20 mA)';
   AIO_2002.___________0030_1 := false;
   AIO_2002.___________0030_2 := false;
   AIO_2002.PARAM_TYPE := 16#02;
   AIO_2002.PARAM_RANGE := 16#02;
   AIO_2002.PARAM_COEF := 16#00;
   AIO_2003.AIO_CODE := 16#2003;
   AIO_2003.___________0020_0 := false;
   AIO_2003.___________0010_2 := false;
   AIO_2003.RAW_MIN := 0;
   AIO_2003.RAW_MAX := 27648;
   AIO_2003.RAW_NAME := 'Current - 4 wire (4 mA to 20 mA)';
   AIO_2003.___________0030_1 := false;
   AIO_2003.___________0030_2 := false;
   AIO_2003.PARAM_TYPE := 16#02;
   AIO_2003.PARAM_RANGE := 16#03;
   AIO_2003.PARAM_COEF := 16#00;
   AIO_2004.AIO_CODE := 16#2004;
   AIO_2004.___________0020_0 := false;
   AIO_2004.___________0010_2 := false;
   AIO_2004.RAW_MIN := -27648;
   AIO_2004.RAW_MAX := 27648;
   AIO_2004.RAW_NAME := 'Current - 4 wire (-20 mA to +20 mA)';
   AIO_2004.___________0030_1 := false;
   AIO_2004.___________0030_2 := false;
   AIO_2004.PARAM_TYPE := 16#02;
   AIO_2004.PARAM_RANGE := 16#04;
   AIO_2004.PARAM_COEF := 16#00;
   AIO_3003.AIO_CODE := 16#3003;
   AIO_3003.___________0020_0 := false;
   AIO_3003.___________0010_2 := false;
   AIO_3003.RAW_MIN := 0;
   AIO_3003.RAW_MAX := 27648;
   AIO_3003.RAW_NAME := 'Current - 2 wire (4 mA to 20 mA)';
   AIO_3003.___________0030_1 := false;
   AIO_3003.___________0030_2 := false;
   AIO_3003.PARAM_TYPE := 16#03;
   AIO_3003.PARAM_RANGE := 16#03;
   AIO_3003.PARAM_COEF := 16#00;
   AIO_4001.AIO_CODE := 16#4001;
   AIO_4001.___________0020_0 := false;
   AIO_4001.___________0010_2 := false;
   AIO_4001.RAW_MIN := 0;
   AIO_4001.RAW_MAX := 27648;
   AIO_4001.RAW_NAME := 'Resistance - 4 wire (150 Ohm)';
   AIO_4001.___________0030_1 := false;
   AIO_4001.___________0030_2 := false;
   AIO_4001.PARAM_TYPE := 16#04;
   AIO_4001.PARAM_RANGE := 16#01;
   AIO_4001.PARAM_COEF := 16#00;
   AIO_4002.AIO_CODE := 16#4002;
   AIO_4002.___________0020_0 := false;
   AIO_4002.___________0010_2 := false;
   AIO_4002.RAW_MIN := 0;
   AIO_4002.RAW_MAX := 27648;
   AIO_4002.RAW_NAME := 'Resistance - 4 wire (300 Ohm)';
   AIO_4002.___________0030_1 := false;
   AIO_4002.___________0030_2 := false;
   AIO_4002.PARAM_TYPE := 16#04;
   AIO_4002.PARAM_RANGE := 16#02;
   AIO_4002.PARAM_COEF := 16#00;
   AIO_4003.AIO_CODE := 16#4003;
   AIO_4003.___________0020_0 := false;
   AIO_4003.___________0010_2 := false;
   AIO_4003.RAW_MIN := 0;
   AIO_4003.RAW_MAX := 27648;
   AIO_4003.RAW_NAME := 'Resistance - 4 wire (600 Ohm)';
   AIO_4003.___________0030_1 := false;
   AIO_4003.___________0030_2 := false;
   AIO_4003.PARAM_TYPE := 16#04;
   AIO_4003.PARAM_RANGE := 16#03;
   AIO_4003.PARAM_COEF := 16#00;
   AIO_4005.AIO_CODE := 16#4005;
   AIO_4005.___________0020_0 := false;
   AIO_4005.___________0010_2 := false;
   AIO_4005.RAW_MIN := 0;
   AIO_4005.RAW_MAX := 27648;
   AIO_4005.RAW_NAME := 'Resistance - 4 wire (6000 Ohm)';
   AIO_4005.___________0030_1 := false;
   AIO_4005.___________0030_2 := false;
   AIO_4005.PARAM_TYPE := 16#04;
   AIO_4005.PARAM_RANGE := 16#05;
   AIO_4005.PARAM_COEF := 16#00;
   AIO_5001.AIO_CODE := 16#5001;
   AIO_5001.___________0020_0 := false;
   AIO_5001.___________0010_2 := false;
   AIO_5001.RAW_MIN := 0;
   AIO_5001.RAW_MAX := 27648;
   AIO_5001.RAW_NAME := 'Resistance - 3 wire (150 Ohm)';
   AIO_5001.___________0030_1 := false;
   AIO_5001.___________0030_2 := false;
   AIO_5001.PARAM_TYPE := 16#05;
   AIO_5001.PARAM_RANGE := 16#01;
   AIO_5001.PARAM_COEF := 16#00;
   AIO_5002.AIO_CODE := 16#5002;
   AIO_5002.___________0020_0 := false;
   AIO_5002.___________0010_2 := false;
   AIO_5002.RAW_MIN := 0;
   AIO_5002.RAW_MAX := 27648;
   AIO_5002.RAW_NAME := 'Resistance - 3 wire (300 Ohm)';
   AIO_5002.___________0030_1 := false;
   AIO_5002.___________0030_2 := false;
   AIO_5002.PARAM_TYPE := 16#05;
   AIO_5002.PARAM_RANGE := 16#02;
   AIO_5002.PARAM_COEF := 16#00;
   AIO_5003.AIO_CODE := 16#5003;
   AIO_5003.___________0020_0 := false;
   AIO_5003.___________0010_2 := false;
   AIO_5003.RAW_MIN := 0;
   AIO_5003.RAW_MAX := 27648;
   AIO_5003.RAW_NAME := 'Resistance - 3 wire (600 Ohm)';
   AIO_5003.___________0030_1 := false;
   AIO_5003.___________0030_2 := false;
   AIO_5003.PARAM_TYPE := 16#05;
   AIO_5003.PARAM_RANGE := 16#03;
   AIO_5003.PARAM_COEF := 16#00;
   AIO_5005.AIO_CODE := 16#5005;
   AIO_5005.___________0020_0 := false;
   AIO_5005.___________0010_2 := false;
   AIO_5005.RAW_MIN := 0;
   AIO_5005.RAW_MAX := 27648;
   AIO_5005.RAW_NAME := 'Resistance - 3 wire (6000 Ohm)';
   AIO_5005.___________0030_1 := false;
   AIO_5005.___________0030_2 := false;
   AIO_5005.PARAM_TYPE := 16#05;
   AIO_5005.PARAM_RANGE := 16#05;
   AIO_5005.PARAM_COEF := 16#00;
   AIO_6001.AIO_CODE := 16#6001;
   AIO_6001.___________0020_0 := false;
   AIO_6001.___________0010_2 := false;
   AIO_6001.RAW_MIN := 0;
   AIO_6001.RAW_MAX := 27648;
   AIO_6001.RAW_NAME := 'Resistance - 2 wire (150 Ohm)';
   AIO_6001.___________0030_1 := false;
   AIO_6001.___________0030_2 := false;
   AIO_6001.PARAM_TYPE := 16#06;
   AIO_6001.PARAM_RANGE := 16#01;
   AIO_6001.PARAM_COEF := 16#00;
   AIO_6002.AIO_CODE := 16#6002;
   AIO_6002.___________0020_0 := false;
   AIO_6002.___________0010_2 := false;
   AIO_6002.RAW_MIN := 0;
   AIO_6002.RAW_MAX := 27648;
   AIO_6002.RAW_NAME := 'Resistance - 2 wire (300 Ohm)';
   AIO_6002.___________0030_1 := false;
   AIO_6002.___________0030_2 := false;
   AIO_6002.PARAM_TYPE := 16#06;
   AIO_6002.PARAM_RANGE := 16#02;
   AIO_6002.PARAM_COEF := 16#00;
   AIO_6003.AIO_CODE := 16#6003;
   AIO_6003.___________0020_0 := false;
   AIO_6003.___________0010_2 := false;
   AIO_6003.RAW_MIN := 0;
   AIO_6003.RAW_MAX := 27648;
   AIO_6003.RAW_NAME := 'Resistance - 2 wire (600 Ohm)';
   AIO_6003.___________0030_1 := false;
   AIO_6003.___________0030_2 := false;
   AIO_6003.PARAM_TYPE := 16#06;
   AIO_6003.PARAM_RANGE := 16#03;
   AIO_6003.PARAM_COEF := 16#00;
   AIO_6005.AIO_CODE := 16#6005;
   AIO_6005.___________0020_0 := false;
   AIO_6005.___________0010_2 := false;
   AIO_6005.RAW_MIN := 0;
   AIO_6005.RAW_MAX := 27648;
   AIO_6005.RAW_NAME := 'Resistance - 2 wire (6000 Ohm)';
   AIO_6005.___________0030_1 := false;
   AIO_6005.___________0030_2 := false;
   AIO_6005.PARAM_TYPE := 16#06;
   AIO_6005.PARAM_RANGE := 16#05;
   AIO_6005.PARAM_COEF := 16#00;
   AIO_600F.AIO_CODE := 16#600F;
   AIO_600F.___________0020_0 := false;
   AIO_600F.___________0010_2 := false;
   AIO_600F.RAW_MIN := 0;
   AIO_600F.RAW_MAX := 27648;
   AIO_600F.RAW_NAME := 'Resistance - 2 wire (PTC)';
   AIO_600F.___________0030_1 := false;
   AIO_600F.___________0030_2 := false;
   AIO_600F.PARAM_TYPE := 16#06;
   AIO_600F.PARAM_RANGE := 16#0F;
   AIO_600F.PARAM_COEF := 16#00;
   AIO_7B0E.AIO_CODE := 16#7B0E;
   AIO_7B0E.___________0020_0 := false;
   AIO_7B0E.___________0010_2 := false;
   AIO_7B0E.RAW_MIN := -5000;
   AIO_7B0E.RAW_MAX := 15000;
   AIO_7B0E.RAW_NAME := 'Thermal Resistance - 4 wire (Cu10 climate - 426)';
   AIO_7B0E.___________0030_1 := false;
   AIO_7B0E.___________0030_2 := false;
   AIO_7B0E.PARAM_TYPE := 16#07;
   AIO_7B0E.PARAM_RANGE := 16#0E;
   AIO_7B0E.PARAM_COEF := 16#0B;
   AIO_7B0E.VALUE_COEF := 0.00426;
   AIO_7C0E.AIO_CODE := 16#7C0E;
   AIO_7C0E.___________0020_0 := false;
   AIO_7C0E.___________0010_2 := false;
   AIO_7C0E.RAW_MIN := -5000;
   AIO_7C0E.RAW_MAX := 15000;
   AIO_7C0E.RAW_NAME := 'Thermal Resistance - 4 wire (Cu10 climate - 427)';
   AIO_7C0E.___________0030_1 := false;
   AIO_7C0E.___________0030_2 := false;
   AIO_7C0E.PARAM_TYPE := 16#07;
   AIO_7C0E.PARAM_RANGE := 16#0E;
   AIO_7C0E.PARAM_COEF := 16#0C;
   AIO_7C0E.VALUE_COEF := 0.00427;
   AIO_7D0E.AIO_CODE := 16#7D0E;
   AIO_7D0E.___________0020_0 := false;
   AIO_7D0E.___________0010_2 := false;
   AIO_7D0E.RAW_MIN := -1800;
   AIO_7D0E.RAW_MAX := 15000;
   AIO_7D0E.RAW_NAME := 'Thermal Resistance - 4 wire (Cu10 climate - 428)';
   AIO_7D0E.___________0030_1 := false;
   AIO_7D0E.___________0030_2 := false;
   AIO_7D0E.PARAM_TYPE := 16#07;
   AIO_7D0E.PARAM_RANGE := 16#0E;
   AIO_7D0E.PARAM_COEF := 16#0D;
   AIO_7D0E.VALUE_COEF := 0.00428;
   AIO_7B0F.AIO_CODE := 16#7B0F;
   AIO_7B0F.___________0020_0 := false;
   AIO_7B0F.___________0010_2 := false;
   AIO_7B0F.RAW_MIN := -500;
   AIO_7B0F.RAW_MAX := 2000;
   AIO_7B0F.RAW_NAME := 'Thermal Resistance - 4 wire (Cu10 standard - 426)';
   AIO_7B0F.___________0030_1 := false;
   AIO_7B0F.___________0030_2 := false;
   AIO_7B0F.PARAM_TYPE := 16#07;
   AIO_7B0F.PARAM_RANGE := 16#0F;
   AIO_7B0F.PARAM_COEF := 16#0B;
   AIO_7B0F.VALUE_COEF := 0.00426;
   AIO_7C0F.AIO_CODE := 16#7C0F;
   AIO_7C0F.___________0020_0 := false;
   AIO_7C0F.___________0010_2 := false;
   AIO_7C0F.RAW_MIN := -2000;
   AIO_7C0F.RAW_MAX := 2600;
   AIO_7C0F.RAW_NAME := 'Thermal Resistance - 4 wire (Cu10 standard - 427)';
   AIO_7C0F.___________0030_1 := false;
   AIO_7C0F.___________0030_2 := false;
   AIO_7C0F.PARAM_TYPE := 16#07;
   AIO_7C0F.PARAM_RANGE := 16#0F;
   AIO_7C0F.PARAM_COEF := 16#0C;
   AIO_7C0F.VALUE_COEF := 0.00427;
   AIO_7D0F.AIO_CODE := 16#7D0F;
   AIO_7D0F.___________0020_0 := false;
   AIO_7D0F.___________0010_2 := false;
   AIO_7D0F.RAW_MIN := -1800;
   AIO_7D0F.RAW_MAX := 2000;
   AIO_7D0F.RAW_NAME := 'Thermal Resistance - 4 wire (Cu10 standard - 428)';
   AIO_7D0F.___________0030_1 := false;
   AIO_7D0F.___________0030_2 := false;
   AIO_7D0F.PARAM_TYPE := 16#07;
   AIO_7D0F.PARAM_RANGE := 16#0F;
   AIO_7D0F.PARAM_COEF := 16#0D;
   AIO_7D0F.VALUE_COEF := 0.00428;
   AIO_7B19.AIO_CODE := 16#7B19;
   AIO_7B19.___________0020_0 := false;
   AIO_7B19.___________0010_2 := false;
   AIO_7B19.RAW_MIN := -5000;
   AIO_7B19.RAW_MAX := 15000;
   AIO_7B19.RAW_NAME := 'Thermal Resistance - 4 wire (Cu50 climate - 426)';
   AIO_7B19.___________0030_1 := false;
   AIO_7B19.___________0030_2 := false;
   AIO_7B19.PARAM_TYPE := 16#07;
   AIO_7B19.PARAM_RANGE := 16#19;
   AIO_7B19.PARAM_COEF := 16#0B;
   AIO_7B19.VALUE_COEF := 0.00426;
   AIO_7C19.AIO_CODE := 16#7C19;
   AIO_7C19.___________0020_0 := false;
   AIO_7C19.___________0010_2 := false;
   AIO_7C19.RAW_MIN := -5000;
   AIO_7C19.RAW_MAX := 15000;
   AIO_7C19.RAW_NAME := 'Thermal Resistance - 4 wire (Cu50 climate - 427)';
   AIO_7C19.___________0030_1 := false;
   AIO_7C19.___________0030_2 := false;
   AIO_7C19.PARAM_TYPE := 16#07;
   AIO_7C19.PARAM_RANGE := 16#19;
   AIO_7C19.PARAM_COEF := 16#0C;
   AIO_7C19.VALUE_COEF := 0.00427;
   AIO_7D19.AIO_CODE := 16#7D19;
   AIO_7D19.___________0020_0 := false;
   AIO_7D19.___________0010_2 := false;
   AIO_7D19.RAW_MIN := -5000;
   AIO_7D19.RAW_MAX := 15000;
   AIO_7D19.RAW_NAME := 'Thermal Resistance - 4 wire (Cu50 climate - 428)';
   AIO_7D19.___________0030_1 := false;
   AIO_7D19.___________0030_2 := false;
   AIO_7D19.PARAM_TYPE := 16#07;
   AIO_7D19.PARAM_RANGE := 16#19;
   AIO_7D19.PARAM_COEF := 16#0D;
   AIO_7D19.VALUE_COEF := 0.00428;
   AIO_7B18.AIO_CODE := 16#7B18;
   AIO_7B18.___________0020_0 := false;
   AIO_7B18.___________0010_2 := false;
   AIO_7B18.RAW_MIN := -500;
   AIO_7B18.RAW_MAX := 2000;
   AIO_7B18.RAW_NAME := 'Thermal Resistance - 4 wire (Cu50 standard - 426)';
   AIO_7B18.___________0030_1 := false;
   AIO_7B18.___________0030_2 := false;
   AIO_7B18.PARAM_TYPE := 16#07;
   AIO_7B18.PARAM_RANGE := 16#18;
   AIO_7B18.PARAM_COEF := 16#0B;
   AIO_7B18.VALUE_COEF := 0.00426;
   AIO_7C18.AIO_CODE := 16#7C18;
   AIO_7C18.___________0020_0 := false;
   AIO_7C18.___________0010_2 := false;
   AIO_7C18.RAW_MIN := -2000;
   AIO_7C18.RAW_MAX := 2600;
   AIO_7C18.RAW_NAME := 'Thermal Resistance - 4 wire (Cu50 standard - 427)';
   AIO_7C18.___________0030_1 := false;
   AIO_7C18.___________0030_2 := false;
   AIO_7C18.PARAM_TYPE := 16#07;
   AIO_7C18.PARAM_RANGE := 16#18;
   AIO_7C18.PARAM_COEF := 16#0C;
   AIO_7C18.VALUE_COEF := 0.00427;
   AIO_7D18.AIO_CODE := 16#7D18;
   AIO_7D18.___________0020_0 := false;
   AIO_7D18.___________0010_2 := false;
   AIO_7D18.RAW_MIN := -1800;
   AIO_7D18.RAW_MAX := 2000;
   AIO_7D18.RAW_NAME := 'Thermal Resistance - 4 wire (Cu50 standard - 428)';
   AIO_7D18.___________0030_1 := false;
   AIO_7D18.___________0030_2 := false;
   AIO_7D18.PARAM_TYPE := 16#07;
   AIO_7D18.PARAM_RANGE := 16#18;
   AIO_7D18.PARAM_COEF := 16#0D;
   AIO_7D18.VALUE_COEF := 0.00428;
   AIO_7B1B.AIO_CODE := 16#7B1B;
   AIO_7B1B.___________0020_0 := false;
   AIO_7B1B.___________0010_2 := false;
   AIO_7B1B.RAW_MIN := -5000;
   AIO_7B1B.RAW_MAX := 15000;
   AIO_7B1B.RAW_NAME := 'Thermal Resistance - 4 wire (Cu100 climate - 426)';
   AIO_7B1B.___________0030_1 := false;
   AIO_7B1B.___________0030_2 := false;
   AIO_7B1B.PARAM_TYPE := 16#07;
   AIO_7B1B.PARAM_RANGE := 16#1B;
   AIO_7B1B.PARAM_COEF := 16#0B;
   AIO_7B1B.VALUE_COEF := 0.00426;
   AIO_7C1B.AIO_CODE := 16#7C1B;
   AIO_7C1B.___________0020_0 := false;
   AIO_7C1B.___________0010_2 := false;
   AIO_7C1B.RAW_MIN := -5000;
   AIO_7C1B.RAW_MAX := 15000;
   AIO_7C1B.RAW_NAME := 'Thermal Resistance - 4 wire (Cu100 climate - 427)';
   AIO_7C1B.___________0030_1 := false;
   AIO_7C1B.___________0030_2 := false;
   AIO_7C1B.PARAM_TYPE := 16#07;
   AIO_7C1B.PARAM_RANGE := 16#1B;
   AIO_7C1B.PARAM_COEF := 16#0C;
   AIO_7C1B.VALUE_COEF := 0.00427;
   AIO_7D1B.AIO_CODE := 16#7D1B;
   AIO_7D1B.___________0020_0 := false;
   AIO_7D1B.___________0010_2 := false;
   AIO_7D1B.RAW_MIN := -5000;
   AIO_7D1B.RAW_MAX := 15000;
   AIO_7D1B.RAW_NAME := 'Thermal Resistance - 4 wire (Cu100 climate - 428)';
   AIO_7D1B.___________0030_1 := false;
   AIO_7D1B.___________0030_2 := false;
   AIO_7D1B.PARAM_TYPE := 16#07;
   AIO_7D1B.PARAM_RANGE := 16#1B;
   AIO_7D1B.PARAM_COEF := 16#0D;
   AIO_7D1B.VALUE_COEF := 0.00428;
   AIO_7B1A.AIO_CODE := 16#7B1A;
   AIO_7B1A.___________0020_0 := false;
   AIO_7B1A.___________0010_2 := false;
   AIO_7B1A.RAW_MIN := -500;
   AIO_7B1A.RAW_MAX := 2000;
   AIO_7B1A.RAW_NAME := 'Thermal Resistance - 4 wire (Cu100 standard - 426)';
   AIO_7B1A.___________0030_1 := false;
   AIO_7B1A.___________0030_2 := false;
   AIO_7B1A.PARAM_TYPE := 16#07;
   AIO_7B1A.PARAM_RANGE := 16#1A;
   AIO_7B1A.PARAM_COEF := 16#0B;
   AIO_7B1A.VALUE_COEF := 0.00426;
   AIO_7C1A.AIO_CODE := 16#7C1A;
   AIO_7C1A.___________0020_0 := false;
   AIO_7C1A.___________0010_2 := false;
   AIO_7C1A.RAW_MIN := -2000;
   AIO_7C1A.RAW_MAX := 2600;
   AIO_7C1A.RAW_NAME := 'Thermal Resistance - 4 wire (Cu100 standard - 427)';
   AIO_7C1A.___________0030_1 := false;
   AIO_7C1A.___________0030_2 := false;
   AIO_7C1A.PARAM_TYPE := 16#07;
   AIO_7C1A.PARAM_RANGE := 16#1A;
   AIO_7C1A.PARAM_COEF := 16#0C;
   AIO_7C1A.VALUE_COEF := 0.00427;
   AIO_7D1A.AIO_CODE := 16#7D1A;
   AIO_7D1A.___________0020_0 := false;
   AIO_7D1A.___________0010_2 := false;
   AIO_7D1A.RAW_MIN := -1800;
   AIO_7D1A.RAW_MAX := 2000;
   AIO_7D1A.RAW_NAME := 'Thermal Resistance - 4 wire (Cu100 standard - 428)';
   AIO_7D1A.___________0030_1 := false;
   AIO_7D1A.___________0030_2 := false;
   AIO_7D1A.PARAM_TYPE := 16#07;
   AIO_7D1A.PARAM_RANGE := 16#1A;
   AIO_7D1A.PARAM_COEF := 16#0D;
   AIO_7D1A.VALUE_COEF := 0.00428;
   AIO_7A1D.AIO_CODE := 16#7A1D;
   AIO_7A1D.___________0020_0 := false;
   AIO_7A1D.___________0010_2 := false;
   AIO_7A1D.RAW_MIN := -6000;
   AIO_7A1D.RAW_MAX := 13000;
   AIO_7A1D.RAW_NAME := 'Thermal Resistance - 4 wire (LG-Ni1000 climate - 500)';
   AIO_7A1D.___________0030_1 := false;
   AIO_7A1D.___________0030_2 := false;
   AIO_7A1D.PARAM_TYPE := 16#07;
   AIO_7A1D.PARAM_RANGE := 16#1D;
   AIO_7A1D.PARAM_COEF := 16#0A;
   AIO_7A1D.VALUE_COEF := 0.005;
   AIO_7A1C.AIO_CODE := 16#7A1C;
   AIO_7A1C.___________0020_0 := false;
   AIO_7A1C.___________0010_2 := false;
   AIO_7A1C.RAW_MIN := -600;
   AIO_7A1C.RAW_MAX := 2500;
   AIO_7A1C.RAW_NAME := 'Thermal Resistance - 4 wire (LG-Ni1000 standard - 500)';
   AIO_7A1C.___________0030_1 := false;
   AIO_7A1C.___________0030_2 := false;
   AIO_7A1C.PARAM_TYPE := 16#07;
   AIO_7A1C.PARAM_RANGE := 16#1C;
   AIO_7A1C.PARAM_COEF := 16#0A;
   AIO_7A1C.VALUE_COEF := 0.005;
   AIO_771F.AIO_CODE := 16#771F;
   AIO_771F.___________0020_0 := false;
   AIO_771F.___________0010_2 := false;
   AIO_771F.RAW_MIN := -6000;
   AIO_771F.RAW_MAX := 13000;
   AIO_771F.RAW_NAME := 'Thermal Resistance - 4 wire (Ni10 climate - 617)';
   AIO_771F.___________0030_1 := false;
   AIO_771F.___________0030_2 := false;
   AIO_771F.PARAM_TYPE := 16#07;
   AIO_771F.PARAM_RANGE := 16#1F;
   AIO_771F.PARAM_COEF := 16#07;
   AIO_771F.VALUE_COEF := 0.00617;
   AIO_781F.AIO_CODE := 16#781F;
   AIO_781F.___________0020_0 := false;
   AIO_781F.___________0010_2 := false;
   AIO_781F.RAW_MIN := -6000;
   AIO_781F.RAW_MAX := 13000;
   AIO_781F.RAW_NAME := 'Thermal Resistance - 4 wire (Ni10 climate - 618)';
   AIO_781F.___________0030_1 := false;
   AIO_781F.___________0030_2 := false;
   AIO_781F.PARAM_TYPE := 16#07;
   AIO_781F.PARAM_RANGE := 16#1F;
   AIO_781F.PARAM_COEF := 16#08;
   AIO_781F.VALUE_COEF := 0.00618;
   AIO_791F.AIO_CODE := 16#791F;
   AIO_791F.___________0020_0 := false;
   AIO_791F.___________0010_2 := false;
   AIO_791F.RAW_MIN := -6000;
   AIO_791F.RAW_MAX := 13000;
   AIO_791F.RAW_NAME := 'Thermal Resistance - 4 wire (Ni10 climate - 672)';
   AIO_791F.___________0030_1 := false;
   AIO_791F.___________0030_2 := false;
   AIO_791F.PARAM_TYPE := 16#07;
   AIO_791F.PARAM_RANGE := 16#1F;
   AIO_791F.PARAM_COEF := 16#09;
   AIO_791F.VALUE_COEF := 0.00672;
   AIO_771E.AIO_CODE := 16#771E;
   AIO_771E.___________0020_0 := false;
   AIO_771E.___________0010_2 := false;
   AIO_771E.RAW_MIN := -600;
   AIO_771E.RAW_MAX := 1800;
   AIO_771E.RAW_NAME := 'Thermal Resistance - 4 wire (Ni10 standard - 617)';
   AIO_771E.___________0030_1 := false;
   AIO_771E.___________0030_2 := false;
   AIO_771E.PARAM_TYPE := 16#07;
   AIO_771E.PARAM_RANGE := 16#1E;
   AIO_771E.PARAM_COEF := 16#07;
   AIO_771E.VALUE_COEF := 0.00617;
   AIO_781E.AIO_CODE := 16#781E;
   AIO_781E.___________0020_0 := false;
   AIO_781E.___________0010_2 := false;
   AIO_781E.RAW_MIN := -600;
   AIO_781E.RAW_MAX := 2500;
   AIO_781E.RAW_NAME := 'Thermal Resistance - 4 wire (Ni10 standard - 618)';
   AIO_781E.___________0030_1 := false;
   AIO_781E.___________0030_2 := false;
   AIO_781E.PARAM_TYPE := 16#07;
   AIO_781E.PARAM_RANGE := 16#1E;
   AIO_781E.PARAM_COEF := 16#08;
   AIO_781E.VALUE_COEF := 0.00618;
   AIO_791E.AIO_CODE := 16#791E;
   AIO_791E.___________0020_0 := false;
   AIO_791E.___________0010_2 := false;
   AIO_791E.RAW_MIN := -600;
   AIO_791E.RAW_MAX := 2500;
   AIO_791E.RAW_NAME := 'Thermal Resistance - 4 wire (Ni10 standard - 672)';
   AIO_791E.___________0030_1 := false;
   AIO_791E.___________0030_2 := false;
   AIO_791E.PARAM_TYPE := 16#07;
   AIO_791E.PARAM_RANGE := 16#1E;
   AIO_791E.PARAM_COEF := 16#09;
   AIO_791E.VALUE_COEF := 0.00672;
   AIO_770D.AIO_CODE := 16#770D;
   AIO_770D.___________0020_0 := false;
   AIO_770D.___________0010_2 := false;
   AIO_770D.RAW_MIN := -6000;
   AIO_770D.RAW_MAX := 13000;
   AIO_770D.RAW_NAME := 'Thermal Resistance - 4 wire (Ni120 climate - 617)';
   AIO_770D.___________0030_1 := false;
   AIO_770D.___________0030_2 := false;
   AIO_770D.PARAM_TYPE := 16#07;
   AIO_770D.PARAM_RANGE := 16#0D;
   AIO_770D.PARAM_COEF := 16#07;
   AIO_770D.VALUE_COEF := 0.00617;
   AIO_780D.AIO_CODE := 16#780D;
   AIO_780D.___________0020_0 := false;
   AIO_780D.___________0010_2 := false;
   AIO_780D.RAW_MIN := -6000;
   AIO_780D.RAW_MAX := 13000;
   AIO_780D.RAW_NAME := 'Thermal Resistance - 4 wire (Ni120 climate - 618)';
   AIO_780D.___________0030_1 := false;
   AIO_780D.___________0030_2 := false;
   AIO_780D.PARAM_TYPE := 16#07;
   AIO_780D.PARAM_RANGE := 16#0D;
   AIO_780D.PARAM_COEF := 16#08;
   AIO_780D.VALUE_COEF := 0.00618;
   AIO_790D.AIO_CODE := 16#790D;
   AIO_790D.___________0020_0 := false;
   AIO_790D.___________0010_2 := false;
   AIO_790D.RAW_MIN := -6000;
   AIO_790D.RAW_MAX := 13000;
   AIO_790D.RAW_NAME := 'Thermal Resistance - 4 wire (Ni120 climate - 672)';
   AIO_790D.___________0030_1 := false;
   AIO_790D.___________0030_2 := false;
   AIO_790D.PARAM_TYPE := 16#07;
   AIO_790D.PARAM_RANGE := 16#0D;
   AIO_790D.PARAM_COEF := 16#09;
   AIO_790D.VALUE_COEF := 0.00672;
   AIO_770C.AIO_CODE := 16#770C;
   AIO_770C.___________0020_0 := false;
   AIO_770C.___________0010_2 := false;
   AIO_770C.RAW_MIN := -600;
   AIO_770C.RAW_MAX := 1800;
   AIO_770C.RAW_NAME := 'Thermal Resistance - 4 wire (Ni120 standard - 617)';
   AIO_770C.___________0030_1 := false;
   AIO_770C.___________0030_2 := false;
   AIO_770C.PARAM_TYPE := 16#07;
   AIO_770C.PARAM_RANGE := 16#0C;
   AIO_770C.PARAM_COEF := 16#07;
   AIO_770C.VALUE_COEF := 0.00617;
   AIO_780C.AIO_CODE := 16#780C;
   AIO_780C.___________0020_0 := false;
   AIO_780C.___________0010_2 := false;
   AIO_780C.RAW_MIN := -600;
   AIO_780C.RAW_MAX := 2500;
   AIO_780C.RAW_NAME := 'Thermal Resistance - 4 wire (Ni120 standard - 618)';
   AIO_780C.___________0030_1 := false;
   AIO_780C.___________0030_2 := false;
   AIO_780C.PARAM_TYPE := 16#07;
   AIO_780C.PARAM_RANGE := 16#0C;
   AIO_780C.PARAM_COEF := 16#08;
   AIO_780C.VALUE_COEF := 0.00618;
   AIO_790C.AIO_CODE := 16#790C;
   AIO_790C.___________0020_0 := false;
   AIO_790C.___________0010_2 := false;
   AIO_790C.RAW_MIN := -600;
   AIO_790C.RAW_MAX := 2500;
   AIO_790C.RAW_NAME := 'Thermal Resistance - 4 wire (Ni120 standard - 672)';
   AIO_790C.___________0030_1 := false;
   AIO_790C.___________0030_2 := false;
   AIO_790C.PARAM_TYPE := 16#07;
   AIO_790C.PARAM_RANGE := 16#0C;
   AIO_790C.PARAM_COEF := 16#09;
   AIO_790C.VALUE_COEF := 0.00672;
   AIO_7701.AIO_CODE := 16#7701;
   AIO_7701.___________0020_0 := false;
   AIO_7701.___________0010_2 := false;
   AIO_7701.RAW_MIN := -6000;
   AIO_7701.RAW_MAX := 13000;
   AIO_7701.RAW_NAME := 'Thermal Resistance - 4 wire (Ni100 climate - 617)';
   AIO_7701.___________0030_1 := false;
   AIO_7701.___________0030_2 := false;
   AIO_7701.PARAM_TYPE := 16#07;
   AIO_7701.PARAM_RANGE := 16#01;
   AIO_7701.PARAM_COEF := 16#07;
   AIO_7701.VALUE_COEF := 0.00617;
   AIO_7801.AIO_CODE := 16#7801;
   AIO_7801.___________0020_0 := false;
   AIO_7801.___________0010_2 := false;
   AIO_7801.RAW_MIN := -6000;
   AIO_7801.RAW_MAX := 13000;
   AIO_7801.RAW_NAME := 'Thermal Resistance - 4 wire (Ni100 climate - 618)';
   AIO_7801.___________0030_1 := false;
   AIO_7801.___________0030_2 := false;
   AIO_7801.PARAM_TYPE := 16#07;
   AIO_7801.PARAM_RANGE := 16#01;
   AIO_7801.PARAM_COEF := 16#08;
   AIO_7801.VALUE_COEF := 0.00618;
   AIO_7901.AIO_CODE := 16#7901;
   AIO_7901.___________0020_0 := false;
   AIO_7901.___________0010_2 := false;
   AIO_7901.RAW_MIN := -6000;
   AIO_7901.RAW_MAX := 13000;
   AIO_7901.RAW_NAME := 'Thermal Resistance - 4 wire (Ni100 climate - 672)';
   AIO_7901.___________0030_1 := false;
   AIO_7901.___________0030_2 := false;
   AIO_7901.PARAM_TYPE := 16#07;
   AIO_7901.PARAM_RANGE := 16#01;
   AIO_7901.PARAM_COEF := 16#09;
   AIO_7901.VALUE_COEF := 0.00672;
   AIO_7703.AIO_CODE := 16#7703;
   AIO_7703.___________0020_0 := false;
   AIO_7703.___________0010_2 := false;
   AIO_7703.RAW_MIN := -600;
   AIO_7703.RAW_MAX := 1800;
   AIO_7703.RAW_NAME := 'Thermal Resistance - 4 wire (Ni100 standard - 617)';
   AIO_7703.___________0030_1 := false;
   AIO_7703.___________0030_2 := false;
   AIO_7703.PARAM_TYPE := 16#07;
   AIO_7703.PARAM_RANGE := 16#03;
   AIO_7703.PARAM_COEF := 16#07;
   AIO_7703.VALUE_COEF := 0.00617;
   AIO_7803.AIO_CODE := 16#7803;
   AIO_7803.___________0020_0 := false;
   AIO_7803.___________0010_2 := false;
   AIO_7803.RAW_MIN := -600;
   AIO_7803.RAW_MAX := 2500;
   AIO_7803.RAW_NAME := 'Thermal Resistance - 4 wire (Ni100 standard - 618)';
   AIO_7803.___________0030_1 := false;
   AIO_7803.___________0030_2 := false;
   AIO_7803.PARAM_TYPE := 16#07;
   AIO_7803.PARAM_RANGE := 16#03;
   AIO_7803.PARAM_COEF := 16#08;
   AIO_7803.VALUE_COEF := 0.00618;
   AIO_7903.AIO_CODE := 16#7903;
   AIO_7903.___________0020_0 := false;
   AIO_7903.___________0010_2 := false;
   AIO_7903.RAW_MIN := -600;
   AIO_7903.RAW_MAX := 2500;
   AIO_7903.RAW_NAME := 'Thermal Resistance - 4 wire (Ni100 standard - 672)';
   AIO_7903.___________0030_1 := false;
   AIO_7903.___________0030_2 := false;
   AIO_7903.PARAM_TYPE := 16#07;
   AIO_7903.PARAM_RANGE := 16#03;
   AIO_7903.PARAM_COEF := 16#09;
   AIO_7903.VALUE_COEF := 0.00672;
   AIO_7711.AIO_CODE := 16#7711;
   AIO_7711.___________0020_0 := false;
   AIO_7711.___________0010_2 := false;
   AIO_7711.RAW_MIN := -6000;
   AIO_7711.RAW_MAX := 13000;
   AIO_7711.RAW_NAME := 'Thermal Resistance - 4 wire (Ni200 climate - 617)';
   AIO_7711.___________0030_1 := false;
   AIO_7711.___________0030_2 := false;
   AIO_7711.PARAM_TYPE := 16#07;
   AIO_7711.PARAM_RANGE := 16#11;
   AIO_7711.PARAM_COEF := 16#07;
   AIO_7711.VALUE_COEF := 0.00617;
   AIO_7811.AIO_CODE := 16#7811;
   AIO_7811.___________0020_0 := false;
   AIO_7811.___________0010_2 := false;
   AIO_7811.RAW_MIN := -6000;
   AIO_7811.RAW_MAX := 13000;
   AIO_7811.RAW_NAME := 'Thermal Resistance - 4 wire (Ni200 climate - 618)';
   AIO_7811.___________0030_1 := false;
   AIO_7811.___________0030_2 := false;
   AIO_7811.PARAM_TYPE := 16#07;
   AIO_7811.PARAM_RANGE := 16#11;
   AIO_7811.PARAM_COEF := 16#08;
   AIO_7811.VALUE_COEF := 0.00618;
   AIO_7911.AIO_CODE := 16#7911;
   AIO_7911.___________0020_0 := false;
   AIO_7911.___________0010_2 := false;
   AIO_7911.RAW_MIN := -6000;
   AIO_7911.RAW_MAX := 13000;
   AIO_7911.RAW_NAME := 'Thermal Resistance - 4 wire (Ni200 climate - 672)';
   AIO_7911.___________0030_1 := false;
   AIO_7911.___________0030_2 := false;
   AIO_7911.PARAM_TYPE := 16#07;
   AIO_7911.PARAM_RANGE := 16#11;
   AIO_7911.PARAM_COEF := 16#09;
   AIO_7911.VALUE_COEF := 0.00672;
   AIO_7710.AIO_CODE := 16#7710;
   AIO_7710.___________0020_0 := false;
   AIO_7710.___________0010_2 := false;
   AIO_7710.RAW_MIN := -600;
   AIO_7710.RAW_MAX := 1800;
   AIO_7710.RAW_NAME := 'Thermal Resistance - 4 wire (Ni200 standard - 617)';
   AIO_7710.___________0030_1 := false;
   AIO_7710.___________0030_2 := false;
   AIO_7710.PARAM_TYPE := 16#07;
   AIO_7710.PARAM_RANGE := 16#10;
   AIO_7710.PARAM_COEF := 16#07;
   AIO_7710.VALUE_COEF := 0.00617;
   AIO_7810.AIO_CODE := 16#7810;
   AIO_7810.___________0020_0 := false;
   AIO_7810.___________0010_2 := false;
   AIO_7810.RAW_MIN := -600;
   AIO_7810.RAW_MAX := 2500;
   AIO_7810.RAW_NAME := 'Thermal Resistance - 4 wire (Ni200 standard - 618)';
   AIO_7810.___________0030_1 := false;
   AIO_7810.___________0030_2 := false;
   AIO_7810.PARAM_TYPE := 16#07;
   AIO_7810.PARAM_RANGE := 16#10;
   AIO_7810.PARAM_COEF := 16#08;
   AIO_7810.VALUE_COEF := 0.00618;
   AIO_7910.AIO_CODE := 16#7910;
   AIO_7910.___________0020_0 := false;
   AIO_7910.___________0010_2 := false;
   AIO_7910.RAW_MIN := -600;
   AIO_7910.RAW_MAX := 2500;
   AIO_7910.RAW_NAME := 'Thermal Resistance - 4 wire (Ni200 standard - 672)';
   AIO_7910.___________0030_1 := false;
   AIO_7910.___________0030_2 := false;
   AIO_7910.PARAM_TYPE := 16#07;
   AIO_7910.PARAM_RANGE := 16#10;
   AIO_7910.PARAM_COEF := 16#09;
   AIO_7910.VALUE_COEF := 0.00672;
   AIO_7713.AIO_CODE := 16#7713;
   AIO_7713.___________0020_0 := false;
   AIO_7713.___________0010_2 := false;
   AIO_7713.RAW_MIN := -6000;
   AIO_7713.RAW_MAX := 13000;
   AIO_7713.RAW_NAME := 'Thermal Resistance - 4 wire (Ni500 climate - 617)';
   AIO_7713.___________0030_1 := false;
   AIO_7713.___________0030_2 := false;
   AIO_7713.PARAM_TYPE := 16#07;
   AIO_7713.PARAM_RANGE := 16#13;
   AIO_7713.PARAM_COEF := 16#07;
   AIO_7713.VALUE_COEF := 0.00617;
   AIO_7813.AIO_CODE := 16#7813;
   AIO_7813.___________0020_0 := false;
   AIO_7813.___________0010_2 := false;
   AIO_7813.RAW_MIN := -6000;
   AIO_7813.RAW_MAX := 13000;
   AIO_7813.RAW_NAME := 'Thermal Resistance - 4 wire (Ni500 climate - 618)';
   AIO_7813.___________0030_1 := false;
   AIO_7813.___________0030_2 := false;
   AIO_7813.PARAM_TYPE := 16#07;
   AIO_7813.PARAM_RANGE := 16#13;
   AIO_7813.PARAM_COEF := 16#08;
   AIO_7813.VALUE_COEF := 0.00618;
   AIO_7913.AIO_CODE := 16#7913;
   AIO_7913.___________0020_0 := false;
   AIO_7913.___________0010_2 := false;
   AIO_7913.RAW_MIN := -6000;
   AIO_7913.RAW_MAX := 13000;
   AIO_7913.RAW_NAME := 'Thermal Resistance - 4 wire (Ni500 climate - 672)';
   AIO_7913.___________0030_1 := false;
   AIO_7913.___________0030_2 := false;
   AIO_7913.PARAM_TYPE := 16#07;
   AIO_7913.PARAM_RANGE := 16#13;
   AIO_7913.PARAM_COEF := 16#09;
   AIO_7913.VALUE_COEF := 0.00672;
   AIO_7712.AIO_CODE := 16#7712;
   AIO_7712.___________0020_0 := false;
   AIO_7712.___________0010_2 := false;
   AIO_7712.RAW_MIN := -600;
   AIO_7712.RAW_MAX := 1800;
   AIO_7712.RAW_NAME := 'Thermal Resistance - 4 wire (Ni500 standard - 617)';
   AIO_7712.___________0030_1 := false;
   AIO_7712.___________0030_2 := false;
   AIO_7712.PARAM_TYPE := 16#07;
   AIO_7712.PARAM_RANGE := 16#12;
   AIO_7712.PARAM_COEF := 16#07;
   AIO_7712.VALUE_COEF := 0.00617;
   AIO_7812.AIO_CODE := 16#7812;
   AIO_7812.___________0020_0 := false;
   AIO_7812.___________0010_2 := false;
   AIO_7812.RAW_MIN := -600;
   AIO_7812.RAW_MAX := 2500;
   AIO_7812.RAW_NAME := 'Thermal Resistance - 4 wire (Ni500 standard - 618)';
   AIO_7812.___________0030_1 := false;
   AIO_7812.___________0030_2 := false;
   AIO_7812.PARAM_TYPE := 16#07;
   AIO_7812.PARAM_RANGE := 16#12;
   AIO_7812.PARAM_COEF := 16#08;
   AIO_7812.VALUE_COEF := 0.00618;
   AIO_7912.AIO_CODE := 16#7912;
   AIO_7912.___________0020_0 := false;
   AIO_7912.___________0010_2 := false;
   AIO_7912.RAW_MIN := -600;
   AIO_7912.RAW_MAX := 2500;
   AIO_7912.RAW_NAME := 'Thermal Resistance - 4 wire (Ni500 standard - 672)';
   AIO_7912.___________0030_1 := false;
   AIO_7912.___________0030_2 := false;
   AIO_7912.PARAM_TYPE := 16#07;
   AIO_7912.PARAM_RANGE := 16#12;
   AIO_7912.PARAM_COEF := 16#09;
   AIO_7912.VALUE_COEF := 0.00672;
   AIO_770A.AIO_CODE := 16#770A;
   AIO_770A.___________0020_0 := false;
   AIO_770A.___________0010_2 := false;
   AIO_770A.RAW_MIN := -6000;
   AIO_770A.RAW_MAX := 13000;
   AIO_770A.RAW_NAME := 'Thermal Resistance - 4 wire (Ni1000 climate - 617)';
   AIO_770A.___________0030_1 := false;
   AIO_770A.___________0030_2 := false;
   AIO_770A.PARAM_TYPE := 16#07;
   AIO_770A.PARAM_RANGE := 16#0A;
   AIO_770A.PARAM_COEF := 16#07;
   AIO_770A.VALUE_COEF := 0.00617;
   AIO_780A.AIO_CODE := 16#780A;
   AIO_780A.___________0020_0 := false;
   AIO_780A.___________0010_2 := false;
   AIO_780A.RAW_MIN := -6000;
   AIO_780A.RAW_MAX := 13000;
   AIO_780A.RAW_NAME := 'Thermal Resistance - 4 wire (Ni1000 climate - 618)';
   AIO_780A.___________0030_1 := false;
   AIO_780A.___________0030_2 := false;
   AIO_780A.PARAM_TYPE := 16#07;
   AIO_780A.PARAM_RANGE := 16#0A;
   AIO_780A.PARAM_COEF := 16#08;
   AIO_780A.VALUE_COEF := 0.00618;
   AIO_790A.AIO_CODE := 16#790A;
   AIO_790A.___________0020_0 := false;
   AIO_790A.___________0010_2 := false;
   AIO_790A.RAW_MIN := -6000;
   AIO_790A.RAW_MAX := 13000;
   AIO_790A.RAW_NAME := 'Thermal Resistance - 4 wire (Ni1000 climate - 672)';
   AIO_790A.___________0030_1 := false;
   AIO_790A.___________0030_2 := false;
   AIO_790A.PARAM_TYPE := 16#07;
   AIO_790A.PARAM_RANGE := 16#0A;
   AIO_790A.PARAM_COEF := 16#09;
   AIO_790A.VALUE_COEF := 0.00672;
   AIO_7706.AIO_CODE := 16#7706;
   AIO_7706.___________0020_0 := false;
   AIO_7706.___________0010_2 := false;
   AIO_7706.RAW_MIN := -600;
   AIO_7706.RAW_MAX := 1800;
   AIO_7706.RAW_NAME := 'Thermal Resistance - 4 wire (Ni1000 standard - 617)';
   AIO_7706.___________0030_1 := false;
   AIO_7706.___________0030_2 := false;
   AIO_7706.PARAM_TYPE := 16#07;
   AIO_7706.PARAM_RANGE := 16#06;
   AIO_7706.PARAM_COEF := 16#07;
   AIO_7706.VALUE_COEF := 0.00617;
   AIO_7806.AIO_CODE := 16#7806;
   AIO_7806.___________0020_0 := false;
   AIO_7806.___________0010_2 := false;
   AIO_7806.RAW_MIN := -600;
   AIO_7806.RAW_MAX := 2500;
   AIO_7806.RAW_NAME := 'Thermal Resistance - 4 wire (Ni1000 standard - 618)';
   AIO_7806.___________0030_1 := false;
   AIO_7806.___________0030_2 := false;
   AIO_7806.PARAM_TYPE := 16#07;
   AIO_7806.PARAM_RANGE := 16#06;
   AIO_7806.PARAM_COEF := 16#08;
   AIO_7806.VALUE_COEF := 0.00618;
   AIO_7906.AIO_CODE := 16#7906;
   AIO_7906.___________0020_0 := false;
   AIO_7906.___________0010_2 := false;
   AIO_7906.RAW_MIN := -600;
   AIO_7906.RAW_MAX := 2500;
   AIO_7906.RAW_NAME := 'Thermal Resistance - 4 wire (Ni1000 standard - 672)';
   AIO_7906.___________0030_1 := false;
   AIO_7906.___________0030_2 := false;
   AIO_7906.PARAM_TYPE := 16#07;
   AIO_7906.PARAM_RANGE := 16#06;
   AIO_7906.PARAM_COEF := 16#09;
   AIO_7906.VALUE_COEF := 0.00672;
   AIO_7015.AIO_CODE := 16#7015;
   AIO_7015.___________0020_0 := false;
   AIO_7015.___________0010_2 := false;
   AIO_7015.RAW_MIN := -12000;
   AIO_7015.RAW_MAX := 13000;
   AIO_7015.RAW_NAME := 'Thermal Resistance - 4 wire (Pt10 climate - 3851)';
   AIO_7015.___________0030_1 := false;
   AIO_7015.___________0030_2 := false;
   AIO_7015.PARAM_TYPE := 16#07;
   AIO_7015.PARAM_RANGE := 16#15;
   AIO_7015.PARAM_COEF := 16#00;
   AIO_7015.VALUE_COEF := 0.003851;
   AIO_7215.AIO_CODE := 16#7215;
   AIO_7215.___________0020_0 := false;
   AIO_7215.___________0010_2 := false;
   AIO_7215.RAW_MIN := -12000;
   AIO_7215.RAW_MAX := 13000;
   AIO_7215.RAW_NAME := 'Thermal Resistance - 4 wire (Pt10 climate - 3902)';
   AIO_7215.___________0030_1 := false;
   AIO_7215.___________0030_2 := false;
   AIO_7215.PARAM_TYPE := 16#07;
   AIO_7215.PARAM_RANGE := 16#15;
   AIO_7215.PARAM_COEF := 16#02;
   AIO_7215.VALUE_COEF := 0.003902;
   AIO_7515.AIO_CODE := 16#7515;
   AIO_7515.___________0020_0 := false;
   AIO_7515.___________0010_2 := false;
   AIO_7515.RAW_MIN := -12000;
   AIO_7515.RAW_MAX := 13000;
   AIO_7515.RAW_NAME := 'Thermal Resistance - 4 wire (Pt10 climate - 391)';
   AIO_7515.___________0030_1 := false;
   AIO_7515.___________0030_2 := false;
   AIO_7515.PARAM_TYPE := 16#07;
   AIO_7515.PARAM_RANGE := 16#15;
   AIO_7515.PARAM_COEF := 16#05;
   AIO_7515.VALUE_COEF := 0.00391;
   AIO_7115.AIO_CODE := 16#7115;
   AIO_7115.___________0020_0 := false;
   AIO_7115.___________0010_2 := false;
   AIO_7115.RAW_MIN := -12000;
   AIO_7115.RAW_MAX := 13000;
   AIO_7115.RAW_NAME := 'Thermal Resistance - 4 wire (Pt10 climate - 3916)';
   AIO_7115.___________0030_1 := false;
   AIO_7115.___________0030_2 := false;
   AIO_7115.PARAM_TYPE := 16#07;
   AIO_7115.PARAM_RANGE := 16#15;
   AIO_7115.PARAM_COEF := 16#01;
   AIO_7115.VALUE_COEF := 0.003916;
   AIO_7315.AIO_CODE := 16#7315;
   AIO_7315.___________0020_0 := false;
   AIO_7315.___________0010_2 := false;
   AIO_7315.RAW_MIN := -12000;
   AIO_7315.RAW_MAX := 13000;
   AIO_7315.RAW_NAME := 'Thermal Resistance - 4 wire (Pt10 climate - 392)';
   AIO_7315.___________0030_1 := false;
   AIO_7315.___________0030_2 := false;
   AIO_7315.PARAM_TYPE := 16#07;
   AIO_7315.PARAM_RANGE := 16#15;
   AIO_7315.PARAM_COEF := 16#03;
   AIO_7315.VALUE_COEF := 0.00392;
   AIO_7014.AIO_CODE := 16#7014;
   AIO_7014.___________0020_0 := false;
   AIO_7014.___________0010_2 := false;
   AIO_7014.RAW_MIN := -2000;
   AIO_7014.RAW_MAX := 8500;
   AIO_7014.RAW_NAME := 'Thermal Resistance - 4 wire (Pt10 standard - 3851)';
   AIO_7014.___________0030_1 := false;
   AIO_7014.___________0030_2 := false;
   AIO_7014.PARAM_TYPE := 16#07;
   AIO_7014.PARAM_RANGE := 16#14;
   AIO_7014.PARAM_COEF := 16#00;
   AIO_7014.VALUE_COEF := 0.003851;
   AIO_7214.AIO_CODE := 16#7214;
   AIO_7214.___________0020_0 := false;
   AIO_7214.___________0010_2 := false;
   AIO_7214.RAW_MIN := -2000;
   AIO_7214.RAW_MAX := 8500;
   AIO_7214.RAW_NAME := 'Thermal Resistance - 4 wire (Pt10 standard - 3902)';
   AIO_7214.___________0030_1 := false;
   AIO_7214.___________0030_2 := false;
   AIO_7214.PARAM_TYPE := 16#07;
   AIO_7214.PARAM_RANGE := 16#14;
   AIO_7214.PARAM_COEF := 16#02;
   AIO_7214.VALUE_COEF := 0.003902;
   AIO_7514.AIO_CODE := 16#7514;
   AIO_7514.___________0020_0 := false;
   AIO_7514.___________0010_2 := false;
   AIO_7514.RAW_MIN := -2000;
   AIO_7514.RAW_MAX := 8500;
   AIO_7514.RAW_NAME := 'Thermal Resistance - 4 wire (Pt10 standard - 391)';
   AIO_7514.___________0030_1 := false;
   AIO_7514.___________0030_2 := false;
   AIO_7514.PARAM_TYPE := 16#07;
   AIO_7514.PARAM_RANGE := 16#14;
   AIO_7514.PARAM_COEF := 16#05;
   AIO_7514.VALUE_COEF := 0.00391;
   AIO_7114.AIO_CODE := 16#7114;
   AIO_7114.___________0020_0 := false;
   AIO_7114.___________0010_2 := false;
   AIO_7114.RAW_MIN := -2000;
   AIO_7114.RAW_MAX := 8500;
   AIO_7114.RAW_NAME := 'Thermal Resistance - 4 wire (Pt10 standard - 3916)';
   AIO_7114.___________0030_1 := false;
   AIO_7114.___________0030_2 := false;
   AIO_7114.PARAM_TYPE := 16#07;
   AIO_7114.PARAM_RANGE := 16#14;
   AIO_7114.PARAM_COEF := 16#01;
   AIO_7114.VALUE_COEF := 0.003916;
   AIO_7314.AIO_CODE := 16#7314;
   AIO_7314.___________0020_0 := false;
   AIO_7314.___________0010_2 := false;
   AIO_7314.RAW_MIN := -2000;
   AIO_7314.RAW_MAX := 8500;
   AIO_7314.RAW_NAME := 'Thermal Resistance - 4 wire (Pt10 standard - 392)';
   AIO_7314.___________0030_1 := false;
   AIO_7314.___________0030_2 := false;
   AIO_7314.PARAM_TYPE := 16#07;
   AIO_7314.PARAM_RANGE := 16#14;
   AIO_7314.PARAM_COEF := 16#03;
   AIO_7314.VALUE_COEF := 0.00392;
   AIO_7017.AIO_CODE := 16#7017;
   AIO_7017.___________0020_0 := false;
   AIO_7017.___________0010_2 := false;
   AIO_7017.RAW_MIN := -12000;
   AIO_7017.RAW_MAX := 13000;
   AIO_7017.RAW_NAME := 'Thermal Resistance - 4 wire (Pt50 climate - 3851)';
   AIO_7017.___________0030_1 := false;
   AIO_7017.___________0030_2 := false;
   AIO_7017.PARAM_TYPE := 16#07;
   AIO_7017.PARAM_RANGE := 16#17;
   AIO_7017.PARAM_COEF := 16#00;
   AIO_7017.VALUE_COEF := 0.003851;
   AIO_7217.AIO_CODE := 16#7217;
   AIO_7217.___________0020_0 := false;
   AIO_7217.___________0010_2 := false;
   AIO_7217.RAW_MIN := -12000;
   AIO_7217.RAW_MAX := 13000;
   AIO_7217.RAW_NAME := 'Thermal Resistance - 4 wire (Pt50 climate - 3902)';
   AIO_7217.___________0030_1 := false;
   AIO_7217.___________0030_2 := false;
   AIO_7217.PARAM_TYPE := 16#07;
   AIO_7217.PARAM_RANGE := 16#17;
   AIO_7217.PARAM_COEF := 16#02;
   AIO_7217.VALUE_COEF := 0.003902;
   AIO_7517.AIO_CODE := 16#7517;
   AIO_7517.___________0020_0 := false;
   AIO_7517.___________0010_2 := false;
   AIO_7517.RAW_MIN := -12000;
   AIO_7517.RAW_MAX := 13000;
   AIO_7517.RAW_NAME := 'Thermal Resistance - 4 wire (Pt50 climate - 391)';
   AIO_7517.___________0030_1 := false;
   AIO_7517.___________0030_2 := false;
   AIO_7517.PARAM_TYPE := 16#07;
   AIO_7517.PARAM_RANGE := 16#17;
   AIO_7517.PARAM_COEF := 16#05;
   AIO_7517.VALUE_COEF := 0.00391;
   AIO_7117.AIO_CODE := 16#7117;
   AIO_7117.___________0020_0 := false;
   AIO_7117.___________0010_2 := false;
   AIO_7117.RAW_MIN := -12000;
   AIO_7117.RAW_MAX := 13000;
   AIO_7117.RAW_NAME := 'Thermal Resistance - 4 wire (Pt50 climate - 3916)';
   AIO_7117.___________0030_1 := false;
   AIO_7117.___________0030_2 := false;
   AIO_7117.PARAM_TYPE := 16#07;
   AIO_7117.PARAM_RANGE := 16#17;
   AIO_7117.PARAM_COEF := 16#01;
   AIO_7117.VALUE_COEF := 0.003916;
   AIO_7317.AIO_CODE := 16#7317;
   AIO_7317.___________0020_0 := false;
   AIO_7317.___________0010_2 := false;
   AIO_7317.RAW_MIN := -12000;
   AIO_7317.RAW_MAX := 13000;
   AIO_7317.RAW_NAME := 'Thermal Resistance - 4 wire (Pt50 climate - 392)';
   AIO_7317.___________0030_1 := false;
   AIO_7317.___________0030_2 := false;
   AIO_7317.PARAM_TYPE := 16#07;
   AIO_7317.PARAM_RANGE := 16#17;
   AIO_7317.PARAM_COEF := 16#03;
   AIO_7317.VALUE_COEF := 0.00392;
   AIO_7016.AIO_CODE := 16#7016;
   AIO_7016.___________0020_0 := false;
   AIO_7016.___________0010_2 := false;
   AIO_7016.RAW_MIN := -2000;
   AIO_7016.RAW_MAX := 8500;
   AIO_7016.RAW_NAME := 'Thermal Resistance - 4 wire (Pt50 standard - 3851)';
   AIO_7016.___________0030_1 := false;
   AIO_7016.___________0030_2 := false;
   AIO_7016.PARAM_TYPE := 16#07;
   AIO_7016.PARAM_RANGE := 16#16;
   AIO_7016.PARAM_COEF := 16#00;
   AIO_7016.VALUE_COEF := 0.003851;
   AIO_7216.AIO_CODE := 16#7216;
   AIO_7216.___________0020_0 := false;
   AIO_7216.___________0010_2 := false;
   AIO_7216.RAW_MIN := -2000;
   AIO_7216.RAW_MAX := 8500;
   AIO_7216.RAW_NAME := 'Thermal Resistance - 4 wire (Pt50 standard - 3902)';
   AIO_7216.___________0030_1 := false;
   AIO_7216.___________0030_2 := false;
   AIO_7216.PARAM_TYPE := 16#07;
   AIO_7216.PARAM_RANGE := 16#16;
   AIO_7216.PARAM_COEF := 16#02;
   AIO_7216.VALUE_COEF := 0.003902;
   AIO_7516.AIO_CODE := 16#7516;
   AIO_7516.___________0020_0 := false;
   AIO_7516.___________0010_2 := false;
   AIO_7516.RAW_MIN := -2000;
   AIO_7516.RAW_MAX := 8500;
   AIO_7516.RAW_NAME := 'Thermal Resistance - 4 wire (Pt50 standard - 391)';
   AIO_7516.___________0030_1 := false;
   AIO_7516.___________0030_2 := false;
   AIO_7516.PARAM_TYPE := 16#07;
   AIO_7516.PARAM_RANGE := 16#16;
   AIO_7516.PARAM_COEF := 16#05;
   AIO_7516.VALUE_COEF := 0.00391;
   AIO_7116.AIO_CODE := 16#7116;
   AIO_7116.___________0020_0 := false;
   AIO_7116.___________0010_2 := false;
   AIO_7116.RAW_MIN := -2000;
   AIO_7116.RAW_MAX := 8500;
   AIO_7116.RAW_NAME := 'Thermal Resistance - 4 wire (Pt50 standard - 3916)';
   AIO_7116.___________0030_1 := false;
   AIO_7116.___________0030_2 := false;
   AIO_7116.PARAM_TYPE := 16#07;
   AIO_7116.PARAM_RANGE := 16#16;
   AIO_7116.PARAM_COEF := 16#01;
   AIO_7116.VALUE_COEF := 0.003916;
   AIO_7316.AIO_CODE := 16#7316;
   AIO_7316.___________0020_0 := false;
   AIO_7316.___________0010_2 := false;
   AIO_7316.RAW_MIN := -2000;
   AIO_7316.RAW_MAX := 8500;
   AIO_7316.RAW_NAME := 'Thermal Resistance - 4 wire (Pt50 standard - 392)';
   AIO_7316.___________0030_1 := false;
   AIO_7316.___________0030_2 := false;
   AIO_7316.PARAM_TYPE := 16#07;
   AIO_7316.PARAM_RANGE := 16#16;
   AIO_7316.PARAM_COEF := 16#03;
   AIO_7316.VALUE_COEF := 0.00392;
   AIO_7000.AIO_CODE := 16#7000;
   AIO_7000.___________0020_0 := false;
   AIO_7000.___________0010_2 := false;
   AIO_7000.RAW_MIN := -12000;
   AIO_7000.RAW_MAX := 13000;
   AIO_7000.RAW_NAME := 'Thermal Resistance - 4 wire (Pt100 climate - 3851)';
   AIO_7000.___________0030_1 := false;
   AIO_7000.___________0030_2 := false;
   AIO_7000.PARAM_TYPE := 16#07;
   AIO_7000.PARAM_RANGE := 16#00;
   AIO_7000.PARAM_COEF := 16#00;
   AIO_7000.VALUE_COEF := 0.003851;
   AIO_7200.AIO_CODE := 16#7200;
   AIO_7200.___________0020_0 := false;
   AIO_7200.___________0010_2 := false;
   AIO_7200.RAW_MIN := -12000;
   AIO_7200.RAW_MAX := 13000;
   AIO_7200.RAW_NAME := 'Thermal Resistance - 4 wire (Pt100 climate - 3902)';
   AIO_7200.___________0030_1 := false;
   AIO_7200.___________0030_2 := false;
   AIO_7200.PARAM_TYPE := 16#07;
   AIO_7200.PARAM_RANGE := 16#00;
   AIO_7200.PARAM_COEF := 16#02;
   AIO_7200.VALUE_COEF := 0.003902;
   AIO_7500.AIO_CODE := 16#7500;
   AIO_7500.___________0020_0 := false;
   AIO_7500.___________0010_2 := false;
   AIO_7500.RAW_MIN := -12000;
   AIO_7500.RAW_MAX := 13000;
   AIO_7500.RAW_NAME := 'Thermal Resistance - 4 wire (Pt100 climate - 391)';
   AIO_7500.___________0030_1 := false;
   AIO_7500.___________0030_2 := false;
   AIO_7500.PARAM_TYPE := 16#07;
   AIO_7500.PARAM_RANGE := 16#00;
   AIO_7500.PARAM_COEF := 16#05;
   AIO_7500.VALUE_COEF := 0.00391;
   AIO_7100.AIO_CODE := 16#7100;
   AIO_7100.___________0020_0 := false;
   AIO_7100.___________0010_2 := false;
   AIO_7100.RAW_MIN := -12000;
   AIO_7100.RAW_MAX := 13000;
   AIO_7100.RAW_NAME := 'Thermal Resistance - 4 wire (Pt100 climate - 3916)';
   AIO_7100.___________0030_1 := false;
   AIO_7100.___________0030_2 := false;
   AIO_7100.PARAM_TYPE := 16#07;
   AIO_7100.PARAM_RANGE := 16#00;
   AIO_7100.PARAM_COEF := 16#01;
   AIO_7100.VALUE_COEF := 0.003916;
   AIO_7300.AIO_CODE := 16#7300;
   AIO_7300.___________0020_0 := false;
   AIO_7300.___________0010_2 := false;
   AIO_7300.RAW_MIN := -12000;
   AIO_7300.RAW_MAX := 13000;
   AIO_7300.RAW_NAME := 'Thermal Resistance - 4 wire (Pt100 climate - 392)';
   AIO_7300.___________0030_1 := false;
   AIO_7300.___________0030_2 := false;
   AIO_7300.PARAM_TYPE := 16#07;
   AIO_7300.PARAM_RANGE := 16#00;
   AIO_7300.PARAM_COEF := 16#03;
   AIO_7300.VALUE_COEF := 0.00392;
   AIO_7002.AIO_CODE := 16#7002;
   AIO_7002.___________0020_0 := false;
   AIO_7002.___________0010_2 := false;
   AIO_7002.RAW_MIN := -2000;
   AIO_7002.RAW_MAX := 8500;
   AIO_7002.RAW_NAME := 'Thermal Resistance - 4 wire (Pt100 standard - 3851)';
   AIO_7002.___________0030_1 := false;
   AIO_7002.___________0030_2 := false;
   AIO_7002.PARAM_TYPE := 16#07;
   AIO_7002.PARAM_RANGE := 16#02;
   AIO_7002.PARAM_COEF := 16#00;
   AIO_7002.VALUE_COEF := 0.003851;
   AIO_7202.AIO_CODE := 16#7202;
   AIO_7202.___________0020_0 := false;
   AIO_7202.___________0010_2 := false;
   AIO_7202.RAW_MIN := -2000;
   AIO_7202.RAW_MAX := 8500;
   AIO_7202.RAW_NAME := 'Thermal Resistance - 4 wire (Pt100 standard - 3902)';
   AIO_7202.___________0030_1 := false;
   AIO_7202.___________0030_2 := false;
   AIO_7202.PARAM_TYPE := 16#07;
   AIO_7202.PARAM_RANGE := 16#02;
   AIO_7202.PARAM_COEF := 16#02;
   AIO_7202.VALUE_COEF := 0.003902;
   AIO_7502.AIO_CODE := 16#7502;
   AIO_7502.___________0020_0 := false;
   AIO_7502.___________0010_2 := false;
   AIO_7502.RAW_MIN := -2000;
   AIO_7502.RAW_MAX := 8500;
   AIO_7502.RAW_NAME := 'Thermal Resistance - 4 wire (Pt100 standard - 391)';
   AIO_7502.___________0030_1 := false;
   AIO_7502.___________0030_2 := false;
   AIO_7502.PARAM_TYPE := 16#07;
   AIO_7502.PARAM_RANGE := 16#02;
   AIO_7502.PARAM_COEF := 16#05;
   AIO_7502.VALUE_COEF := 0.00391;
   AIO_7102.AIO_CODE := 16#7102;
   AIO_7102.___________0020_0 := false;
   AIO_7102.___________0010_2 := false;
   AIO_7102.RAW_MIN := -2000;
   AIO_7102.RAW_MAX := 8500;
   AIO_7102.RAW_NAME := 'Thermal Resistance - 4 wire (Pt100 standard - 3916)';
   AIO_7102.___________0030_1 := false;
   AIO_7102.___________0030_2 := false;
   AIO_7102.PARAM_TYPE := 16#07;
   AIO_7102.PARAM_RANGE := 16#02;
   AIO_7102.PARAM_COEF := 16#01;
   AIO_7102.VALUE_COEF := 0.003916;
   AIO_7302.AIO_CODE := 16#7302;
   AIO_7302.___________0020_0 := false;
   AIO_7302.___________0010_2 := false;
   AIO_7302.RAW_MIN := -2000;
   AIO_7302.RAW_MAX := 8500;
   AIO_7302.RAW_NAME := 'Thermal Resistance - 4 wire (Pt100 standard - 392)';
   AIO_7302.___________0030_1 := false;
   AIO_7302.___________0030_2 := false;
   AIO_7302.PARAM_TYPE := 16#07;
   AIO_7302.PARAM_RANGE := 16#02;
   AIO_7302.PARAM_COEF := 16#03;
   AIO_7302.VALUE_COEF := 0.00392;
   AIO_7007.AIO_CODE := 16#7007;
   AIO_7007.___________0020_0 := false;
   AIO_7007.___________0010_2 := false;
   AIO_7007.RAW_MIN := -12000;
   AIO_7007.RAW_MAX := 13000;
   AIO_7007.RAW_NAME := 'Thermal Resistance - 4 wire (Pt200 climate - 3851)';
   AIO_7007.___________0030_1 := false;
   AIO_7007.___________0030_2 := false;
   AIO_7007.PARAM_TYPE := 16#07;
   AIO_7007.PARAM_RANGE := 16#07;
   AIO_7007.PARAM_COEF := 16#00;
   AIO_7007.VALUE_COEF := 0.003851;
   AIO_7207.AIO_CODE := 16#7207;
   AIO_7207.___________0020_0 := false;
   AIO_7207.___________0010_2 := false;
   AIO_7207.RAW_MIN := -12000;
   AIO_7207.RAW_MAX := 13000;
   AIO_7207.RAW_NAME := 'Thermal Resistance - 4 wire (Pt200 climate - 3902)';
   AIO_7207.___________0030_1 := false;
   AIO_7207.___________0030_2 := false;
   AIO_7207.PARAM_TYPE := 16#07;
   AIO_7207.PARAM_RANGE := 16#07;
   AIO_7207.PARAM_COEF := 16#02;
   AIO_7207.VALUE_COEF := 0.003902;
   AIO_7507.AIO_CODE := 16#7507;
   AIO_7507.___________0020_0 := false;
   AIO_7507.___________0010_2 := false;
   AIO_7507.RAW_MIN := -12000;
   AIO_7507.RAW_MAX := 13000;
   AIO_7507.RAW_NAME := 'Thermal Resistance - 4 wire (Pt200 climate - 391)';
   AIO_7507.___________0030_1 := false;
   AIO_7507.___________0030_2 := false;
   AIO_7507.PARAM_TYPE := 16#07;
   AIO_7507.PARAM_RANGE := 16#07;
   AIO_7507.PARAM_COEF := 16#05;
   AIO_7507.VALUE_COEF := 0.00391;
   AIO_7107.AIO_CODE := 16#7107;
   AIO_7107.___________0020_0 := false;
   AIO_7107.___________0010_2 := false;
   AIO_7107.RAW_MIN := -12000;
   AIO_7107.RAW_MAX := 13000;
   AIO_7107.RAW_NAME := 'Thermal Resistance - 4 wire (Pt200 climate - 3916)';
   AIO_7107.___________0030_1 := false;
   AIO_7107.___________0030_2 := false;
   AIO_7107.PARAM_TYPE := 16#07;
   AIO_7107.PARAM_RANGE := 16#07;
   AIO_7107.PARAM_COEF := 16#01;
   AIO_7107.VALUE_COEF := 0.003916;
   AIO_7307.AIO_CODE := 16#7307;
   AIO_7307.___________0020_0 := false;
   AIO_7307.___________0010_2 := false;
   AIO_7307.RAW_MIN := -12000;
   AIO_7307.RAW_MAX := 13000;
   AIO_7307.RAW_NAME := 'Thermal Resistance - 4 wire (Pt200 climate - 392)';
   AIO_7307.___________0030_1 := false;
   AIO_7307.___________0030_2 := false;
   AIO_7307.PARAM_TYPE := 16#07;
   AIO_7307.PARAM_RANGE := 16#07;
   AIO_7307.PARAM_COEF := 16#03;
   AIO_7307.VALUE_COEF := 0.00392;
   AIO_700B.AIO_CODE := 16#700B;
   AIO_700B.___________0020_0 := false;
   AIO_700B.___________0010_2 := false;
   AIO_700B.RAW_MIN := -2000;
   AIO_700B.RAW_MAX := 8500;
   AIO_700B.RAW_NAME := 'Thermal Resistance - 4 wire (Pt200 standard - 3851)';
   AIO_700B.___________0030_1 := false;
   AIO_700B.___________0030_2 := false;
   AIO_700B.PARAM_TYPE := 16#07;
   AIO_700B.PARAM_RANGE := 16#0B;
   AIO_700B.PARAM_COEF := 16#00;
   AIO_700B.VALUE_COEF := 0.003851;
   AIO_720B.AIO_CODE := 16#720B;
   AIO_720B.___________0020_0 := false;
   AIO_720B.___________0010_2 := false;
   AIO_720B.RAW_MIN := -2000;
   AIO_720B.RAW_MAX := 8500;
   AIO_720B.RAW_NAME := 'Thermal Resistance - 4 wire (Pt200 standard - 3902)';
   AIO_720B.___________0030_1 := false;
   AIO_720B.___________0030_2 := false;
   AIO_720B.PARAM_TYPE := 16#07;
   AIO_720B.PARAM_RANGE := 16#0B;
   AIO_720B.PARAM_COEF := 16#02;
   AIO_720B.VALUE_COEF := 0.003902;
   AIO_750B.AIO_CODE := 16#750B;
   AIO_750B.___________0020_0 := false;
   AIO_750B.___________0010_2 := false;
   AIO_750B.RAW_MIN := -2000;
   AIO_750B.RAW_MAX := 8500;
   AIO_750B.RAW_NAME := 'Thermal Resistance - 4 wire (Pt200 standard - 391)';
   AIO_750B.___________0030_1 := false;
   AIO_750B.___________0030_2 := false;
   AIO_750B.PARAM_TYPE := 16#07;
   AIO_750B.PARAM_RANGE := 16#0B;
   AIO_750B.PARAM_COEF := 16#05;
   AIO_750B.VALUE_COEF := 0.00391;
   AIO_710B.AIO_CODE := 16#710B;
   AIO_710B.___________0020_0 := false;
   AIO_710B.___________0010_2 := false;
   AIO_710B.RAW_MIN := -2000;
   AIO_710B.RAW_MAX := 8500;
   AIO_710B.RAW_NAME := 'Thermal Resistance - 4 wire (Pt200 standard - 3916)';
   AIO_710B.___________0030_1 := false;
   AIO_710B.___________0030_2 := false;
   AIO_710B.PARAM_TYPE := 16#07;
   AIO_710B.PARAM_RANGE := 16#0B;
   AIO_710B.PARAM_COEF := 16#01;
   AIO_710B.VALUE_COEF := 0.003916;
   AIO_730B.AIO_CODE := 16#730B;
   AIO_730B.___________0020_0 := false;
   AIO_730B.___________0010_2 := false;
   AIO_730B.RAW_MIN := -2000;
   AIO_730B.RAW_MAX := 8500;
   AIO_730B.RAW_NAME := 'Thermal Resistance - 4 wire (Pt200 standard - 392)';
   AIO_730B.___________0030_1 := false;
   AIO_730B.___________0030_2 := false;
   AIO_730B.PARAM_TYPE := 16#07;
   AIO_730B.PARAM_RANGE := 16#0B;
   AIO_730B.PARAM_COEF := 16#03;
   AIO_730B.VALUE_COEF := 0.00392;
   AIO_7008.AIO_CODE := 16#7008;
   AIO_7008.___________0020_0 := false;
   AIO_7008.___________0010_2 := false;
   AIO_7008.RAW_MIN := -12000;
   AIO_7008.RAW_MAX := 13000;
   AIO_7008.RAW_NAME := 'Thermal Resistance - 4 wire (Pt500 climate - 3851)';
   AIO_7008.___________0030_1 := false;
   AIO_7008.___________0030_2 := false;
   AIO_7008.PARAM_TYPE := 16#07;
   AIO_7008.PARAM_RANGE := 16#08;
   AIO_7008.PARAM_COEF := 16#00;
   AIO_7008.VALUE_COEF := 0.003851;
   AIO_7208.AIO_CODE := 16#7208;
   AIO_7208.___________0020_0 := false;
   AIO_7208.___________0010_2 := false;
   AIO_7208.RAW_MIN := -12000;
   AIO_7208.RAW_MAX := 13000;
   AIO_7208.RAW_NAME := 'Thermal Resistance - 4 wire (Pt500 climate - 3902)';
   AIO_7208.___________0030_1 := false;
   AIO_7208.___________0030_2 := false;
   AIO_7208.PARAM_TYPE := 16#07;
   AIO_7208.PARAM_RANGE := 16#08;
   AIO_7208.PARAM_COEF := 16#02;
   AIO_7208.VALUE_COEF := 0.003902;
   AIO_7508.AIO_CODE := 16#7508;
   AIO_7508.___________0020_0 := false;
   AIO_7508.___________0010_2 := false;
   AIO_7508.RAW_MIN := -12000;
   AIO_7508.RAW_MAX := 13000;
   AIO_7508.RAW_NAME := 'Thermal Resistance - 4 wire (Pt500 climate - 391)';
   AIO_7508.___________0030_1 := false;
   AIO_7508.___________0030_2 := false;
   AIO_7508.PARAM_TYPE := 16#07;
   AIO_7508.PARAM_RANGE := 16#08;
   AIO_7508.PARAM_COEF := 16#05;
   AIO_7508.VALUE_COEF := 0.00391;
   AIO_7108.AIO_CODE := 16#7108;
   AIO_7108.___________0020_0 := false;
   AIO_7108.___________0010_2 := false;
   AIO_7108.RAW_MIN := -12000;
   AIO_7108.RAW_MAX := 13000;
   AIO_7108.RAW_NAME := 'Thermal Resistance - 4 wire (Pt500 climate - 3916)';
   AIO_7108.___________0030_1 := false;
   AIO_7108.___________0030_2 := false;
   AIO_7108.PARAM_TYPE := 16#07;
   AIO_7108.PARAM_RANGE := 16#08;
   AIO_7108.PARAM_COEF := 16#01;
   AIO_7108.VALUE_COEF := 0.003916;
   AIO_7308.AIO_CODE := 16#7308;
   AIO_7308.___________0020_0 := false;
   AIO_7308.___________0010_2 := false;
   AIO_7308.RAW_MIN := -12000;
   AIO_7308.RAW_MAX := 13000;
   AIO_7308.RAW_NAME := 'Thermal Resistance - 4 wire (Pt500 climate - 392)';
   AIO_7308.___________0030_1 := false;
   AIO_7308.___________0030_2 := false;
   AIO_7308.PARAM_TYPE := 16#07;
   AIO_7308.PARAM_RANGE := 16#08;
   AIO_7308.PARAM_COEF := 16#03;
   AIO_7308.VALUE_COEF := 0.00392;
   AIO_7004.AIO_CODE := 16#7004;
   AIO_7004.___________0020_0 := false;
   AIO_7004.___________0010_2 := false;
   AIO_7004.RAW_MIN := -2000;
   AIO_7004.RAW_MAX := 8500;
   AIO_7004.RAW_NAME := 'Thermal Resistance - 4 wire (Pt500 standard - 3851)';
   AIO_7004.___________0030_1 := false;
   AIO_7004.___________0030_2 := false;
   AIO_7004.PARAM_TYPE := 16#07;
   AIO_7004.PARAM_RANGE := 16#04;
   AIO_7004.PARAM_COEF := 16#00;
   AIO_7004.VALUE_COEF := 0.003851;
   AIO_7204.AIO_CODE := 16#7204;
   AIO_7204.___________0020_0 := false;
   AIO_7204.___________0010_2 := false;
   AIO_7204.RAW_MIN := -2000;
   AIO_7204.RAW_MAX := 8500;
   AIO_7204.RAW_NAME := 'Thermal Resistance - 4 wire (Pt500 standard - 3902)';
   AIO_7204.___________0030_1 := false;
   AIO_7204.___________0030_2 := false;
   AIO_7204.PARAM_TYPE := 16#07;
   AIO_7204.PARAM_RANGE := 16#04;
   AIO_7204.PARAM_COEF := 16#02;
   AIO_7204.VALUE_COEF := 0.003902;
   AIO_7504.AIO_CODE := 16#7504;
   AIO_7504.___________0020_0 := false;
   AIO_7504.___________0010_2 := false;
   AIO_7504.RAW_MIN := -2000;
   AIO_7504.RAW_MAX := 8500;
   AIO_7504.RAW_NAME := 'Thermal Resistance - 4 wire (Pt500 standard - 391)';
   AIO_7504.___________0030_1 := false;
   AIO_7504.___________0030_2 := false;
   AIO_7504.PARAM_TYPE := 16#07;
   AIO_7504.PARAM_RANGE := 16#04;
   AIO_7504.PARAM_COEF := 16#05;
   AIO_7504.VALUE_COEF := 0.00391;
   AIO_7104.AIO_CODE := 16#7104;
   AIO_7104.___________0020_0 := false;
   AIO_7104.___________0010_2 := false;
   AIO_7104.RAW_MIN := -2000;
   AIO_7104.RAW_MAX := 8500;
   AIO_7104.RAW_NAME := 'Thermal Resistance - 4 wire (Pt500 standard - 3916)';
   AIO_7104.___________0030_1 := false;
   AIO_7104.___________0030_2 := false;
   AIO_7104.PARAM_TYPE := 16#07;
   AIO_7104.PARAM_RANGE := 16#04;
   AIO_7104.PARAM_COEF := 16#01;
   AIO_7104.VALUE_COEF := 0.003916;
   AIO_7304.AIO_CODE := 16#7304;
   AIO_7304.___________0020_0 := false;
   AIO_7304.___________0010_2 := false;
   AIO_7304.RAW_MIN := -2000;
   AIO_7304.RAW_MAX := 8500;
   AIO_7304.RAW_NAME := 'Thermal Resistance - 4 wire (Pt500 standard - 392)';
   AIO_7304.___________0030_1 := false;
   AIO_7304.___________0030_2 := false;
   AIO_7304.PARAM_TYPE := 16#07;
   AIO_7304.PARAM_RANGE := 16#04;
   AIO_7304.PARAM_COEF := 16#03;
   AIO_7304.VALUE_COEF := 0.00392;
   AIO_7009.AIO_CODE := 16#7009;
   AIO_7009.___________0020_0 := false;
   AIO_7009.___________0010_2 := false;
   AIO_7009.RAW_MIN := -12000;
   AIO_7009.RAW_MAX := 13000;
   AIO_7009.RAW_NAME := 'Thermal Resistance - 4 wire (Pt1000 climate - 3851)';
   AIO_7009.___________0030_1 := false;
   AIO_7009.___________0030_2 := false;
   AIO_7009.PARAM_TYPE := 16#07;
   AIO_7009.PARAM_RANGE := 16#09;
   AIO_7009.PARAM_COEF := 16#00;
   AIO_7009.VALUE_COEF := 0.003851;
   AIO_7209.AIO_CODE := 16#7209;
   AIO_7209.___________0020_0 := false;
   AIO_7209.___________0010_2 := false;
   AIO_7209.RAW_MIN := -12000;
   AIO_7209.RAW_MAX := 13000;
   AIO_7209.RAW_NAME := 'Thermal Resistance - 4 wire (Pt1000 climate - 3902)';
   AIO_7209.___________0030_1 := false;
   AIO_7209.___________0030_2 := false;
   AIO_7209.PARAM_TYPE := 16#07;
   AIO_7209.PARAM_RANGE := 16#09;
   AIO_7209.PARAM_COEF := 16#02;
   AIO_7209.VALUE_COEF := 0.003902;
   AIO_7509.AIO_CODE := 16#7509;
   AIO_7509.___________0020_0 := false;
   AIO_7509.___________0010_2 := false;
   AIO_7509.RAW_MIN := -12000;
   AIO_7509.RAW_MAX := 13000;
   AIO_7509.RAW_NAME := 'Thermal Resistance - 4 wire (Pt1000 climate - 391)';
   AIO_7509.___________0030_1 := false;
   AIO_7509.___________0030_2 := false;
   AIO_7509.PARAM_TYPE := 16#07;
   AIO_7509.PARAM_RANGE := 16#09;
   AIO_7509.PARAM_COEF := 16#05;
   AIO_7509.VALUE_COEF := 0.00391;
   AIO_7109.AIO_CODE := 16#7109;
   AIO_7109.___________0020_0 := false;
   AIO_7109.___________0010_2 := false;
   AIO_7109.RAW_MIN := -12000;
   AIO_7109.RAW_MAX := 13000;
   AIO_7109.RAW_NAME := 'Thermal Resistance - 4 wire (Pt1000 climate - 3916)';
   AIO_7109.___________0030_1 := false;
   AIO_7109.___________0030_2 := false;
   AIO_7109.PARAM_TYPE := 16#07;
   AIO_7109.PARAM_RANGE := 16#09;
   AIO_7109.PARAM_COEF := 16#01;
   AIO_7109.VALUE_COEF := 0.003916;
   AIO_7309.AIO_CODE := 16#7309;
   AIO_7309.___________0020_0 := false;
   AIO_7309.___________0010_2 := false;
   AIO_7309.RAW_MIN := -12000;
   AIO_7309.RAW_MAX := 13000;
   AIO_7309.RAW_NAME := 'Thermal Resistance - 4 wire (Pt1000 climate - 392)';
   AIO_7309.___________0030_1 := false;
   AIO_7309.___________0030_2 := false;
   AIO_7309.PARAM_TYPE := 16#07;
   AIO_7309.PARAM_RANGE := 16#09;
   AIO_7309.PARAM_COEF := 16#03;
   AIO_7309.VALUE_COEF := 0.00392;
   AIO_7005.AIO_CODE := 16#7005;
   AIO_7005.___________0020_0 := false;
   AIO_7005.___________0010_2 := false;
   AIO_7005.RAW_MIN := -2000;
   AIO_7005.RAW_MAX := 8500;
   AIO_7005.RAW_NAME := 'Thermal Resistance - 4 wire (Pt1000 standard - 3851)';
   AIO_7005.___________0030_1 := false;
   AIO_7005.___________0030_2 := false;
   AIO_7005.PARAM_TYPE := 16#07;
   AIO_7005.PARAM_RANGE := 16#05;
   AIO_7005.PARAM_COEF := 16#00;
   AIO_7005.VALUE_COEF := 0.003851;
   AIO_7205.AIO_CODE := 16#7205;
   AIO_7205.___________0020_0 := false;
   AIO_7205.___________0010_2 := false;
   AIO_7205.RAW_MIN := -2000;
   AIO_7205.RAW_MAX := 8500;
   AIO_7205.RAW_NAME := 'Thermal Resistance - 4 wire (Pt1000 standard - 3902)';
   AIO_7205.___________0030_1 := false;
   AIO_7205.___________0030_2 := false;
   AIO_7205.PARAM_TYPE := 16#07;
   AIO_7205.PARAM_RANGE := 16#05;
   AIO_7205.PARAM_COEF := 16#02;
   AIO_7205.VALUE_COEF := 0.003902;
   AIO_7505.AIO_CODE := 16#7505;
   AIO_7505.___________0020_0 := false;
   AIO_7505.___________0010_2 := false;
   AIO_7505.RAW_MIN := -2000;
   AIO_7505.RAW_MAX := 8500;
   AIO_7505.RAW_NAME := 'Thermal Resistance - 4 wire (Pt1000 standard - 391)';
   AIO_7505.___________0030_1 := false;
   AIO_7505.___________0030_2 := false;
   AIO_7505.PARAM_TYPE := 16#07;
   AIO_7505.PARAM_RANGE := 16#05;
   AIO_7505.PARAM_COEF := 16#05;
   AIO_7505.VALUE_COEF := 0.00391;
   AIO_7105.AIO_CODE := 16#7105;
   AIO_7105.___________0020_0 := false;
   AIO_7105.___________0010_2 := false;
   AIO_7105.RAW_MIN := -2000;
   AIO_7105.RAW_MAX := 8500;
   AIO_7105.RAW_NAME := 'Thermal Resistance - 4 wire (Pt1000 standard - 3916)';
   AIO_7105.___________0030_1 := false;
   AIO_7105.___________0030_2 := false;
   AIO_7105.PARAM_TYPE := 16#07;
   AIO_7105.PARAM_RANGE := 16#05;
   AIO_7105.PARAM_COEF := 16#01;
   AIO_7105.VALUE_COEF := 0.003916;
   AIO_7305.AIO_CODE := 16#7305;
   AIO_7305.___________0020_0 := false;
   AIO_7305.___________0010_2 := false;
   AIO_7305.RAW_MIN := -2000;
   AIO_7305.RAW_MAX := 8500;
   AIO_7305.RAW_NAME := 'Thermal Resistance - 4 wire (Pt1000 standard - 392)';
   AIO_7305.___________0030_1 := false;
   AIO_7305.___________0030_2 := false;
   AIO_7305.PARAM_TYPE := 16#07;
   AIO_7305.PARAM_RANGE := 16#05;
   AIO_7305.PARAM_COEF := 16#03;
   AIO_7305.VALUE_COEF := 0.00392;
   "199".AIO_CODE := 101;
   "199".RAW_MIN := -27648;
   "199".RAW_MAX := 27648;
   "199".RAW_NAME := '-10 V to 10 V';
   AIO_8B0E.AIO_CODE := 16#8B0E;
   AIO_8B0E.___________0020_0 := false;
   AIO_8B0E.___________0010_2 := false;
   AIO_8B0E.RAW_MIN := -5000;
   AIO_8B0E.RAW_MAX := 15000;
   AIO_8B0E.RAW_NAME := 'Thermal Resistance - 3-wire (Cu10 climate - 426)';
   AIO_8B0E.___________0030_1 := false;
   AIO_8B0E.___________0030_2 := false;
   AIO_8B0E.PARAM_TYPE := 16#07;
   AIO_8B0E.PARAM_RANGE := 16#0E;
   AIO_8B0E.PARAM_COEF := 16#0B;
   AIO_8B0E.VALUE_COEF := 0.00426;
   AIO_8C0E.AIO_CODE := 16#8C0E;
   AIO_8C0E.___________0020_0 := false;
   AIO_8C0E.___________0010_2 := false;
   AIO_8C0E.RAW_MIN := -5000;
   AIO_8C0E.RAW_MAX := 15000;
   AIO_8C0E.RAW_NAME := 'Thermal Resistance - 3-wire (Cu10 climate - 427)';
